LIN {X -0.331,Y -633.573,Z 342.601,A 0.000,B 0.000,C 90.000,E1 324.276} C_DIS
LIN {X 0.162,Y -638.117,Z 342.593,A 0.000,B 0.000,C 90.000,E1 322.718} C_DIS
LIN {X 0.137,Y -643.220,Z 342.583,A 0.000,B 0.000,C 90.000,E1 320.964} C_DIS
LIN {X 0.220,Y -647.759,Z 342.575,A 0.000,B 0.000,C 90.000,E1 319.461} C_DIS
LIN {X -0.093,Y -652.321,Z 342.567,A 0.000,B 0.000,C 90.000,E1 318.000} C_DIS
LIN {X 0.029,Y -660.222,Z 342.553,A 0.000,B 0.000,C 90.000,E1 315.526} C_DIS
LIN {X 0.410,Y -664.075,Z 342.546,A 0.000,B 0.000,C 90.000,E1 314.271} C_DIS
LIN {X -0.075,Y -667.878,Z 342.539,A 0.000,B 0.000,C 90.000,E1 313.095} C_DIS
LIN {X 0.010,Y -672.343,Z 342.531,A 0.000,B 0.000,C 90.000,E1 311.634} C_DIS
LIN {X 0.178,Y -676.385,Z 342.523,A 0.000,B 0.000,C 90.000,E1 310.172} C_DIS
LIN {X -0.049,Y -679.539,Z 342.517,A 0.000,B 0.000,C 90.000,E1 308.991} C_DIS
LIN {X 0.163,Y -681.944,Z 342.511,A 0.000,B 0.000,C 90.000,E1 308.016} C_DIS
LIN {X -0.404,Y -684.576,Z 342.505,A 0.000,B 0.000,C 90.000,E1 306.870} C_DIS
LIN {X -0.003,Y -686.307,Z 342.499,A 0.000,B 0.000,C 90.000,E1 305.884} C_DIS
LIN {X -0.162,Y -687.495,Z 342.495,A 0.000,B 0.000,C 90.000,E1 305.185} C_DIS
LIN {X 0.079,Y -688.424,Z 342.491,A 0.000,B 0.000,C 90.000,E1 304.452} C_DIS
LIN {X -0.452,Y -689.214,Z 342.488,A 0.000,B 0.000,C 90.000,E1 303.785} C_DIS
LIN {X -0.225,Y -689.609,Z 342.485,A 0.000,B 0.000,C 90.000,E1 303.293} C_DIS
LIN {X 0.216,Y -689.941,Z 342.481,A 0.000,B 0.000,C 90.000,E1 302.546} C_DIS
LIN {X -0.289,Y -689.979,Z 342.477,A 0.000,B 0.000,C 90.000,E1 301.878} C_DIS
LIN {X -0.067,Y -689.884,Z 342.474,A 0.000,B 0.000,C 90.000,E1 301.386} C_DIS
LIN {X -0.349,Y -689.175,Z 342.469,A 0.000,B 0.000,C 90.000,E1 300.463} C_DIS
LIN {X 0.107,Y -688.694,Z 342.466,A 0.000,B 0.000,C 90.000,E1 299.951} C_DIS
LIN {X -0.069,Y -687.718,Z 342.463,A 0.000,B 0.000,C 90.000,E1 299.255} C_DIS
LIN {X 0.000,Y -686.587,Z 342.459,A 0.000,B 0.000,C 90.000,E1 298.537} C_DIS
LIN {X 0.177,Y -684.270,Z 342.452,A 0.000,B 0.000,C 90.000,E1 297.334} C_DIS
LIN {X -0.067,Y -681.100,Z 342.444,A 0.000,B 0.000,C 90.000,E1 295.924} C_DIS
LIN {X 0.042,Y -678.136,Z 342.437,A 0.000,B 0.000,C 90.000,E1 294.719} C_DIS
LIN {X 0.274,Y -674.479,Z 342.429,A 0.000,B 0.000,C 90.000,E1 293.259} C_DIS
LIN {X -0.100,Y -670.508,Z 342.421,A 0.000,B 0.000,C 90.000,E1 291.844} C_DIS
LIN {X 0.164,Y -664.072,Z 342.408,A 0.000,B 0.000,C 90.000,E1 289.396} C_DIS
LIN {X -0.126,Y -657.475,Z 342.393,A 0.000,B 0.000,C 90.000,E1 286.732} C_DIS
LIN {X -0.104,Y -653.677,Z 342.383,A 0.000,B 0.000,C 90.000,E1 285.009} C_DIS
LIN {X -0.081,Y -648.752,Z 342.370,A 0.000,B 0.000,C 90.000,E1 282.535} C_DIS
LIN {X 0.182,Y -643.588,Z 342.350,A 0.000,B 0.000,C 90.000,E1 279.029} C_DIS
LIN {X 0.176,Y -640.607,Z 342.334,A 0.000,B 0.000,C 90.000,E1 276.030} C_DIS
LIN {X -0.117,Y -639.523,Z 342.324,A 0.000,B 0.000,C 90.000,E1 274.302} C_DIS
LIN {X -0.028,Y -638.474,Z 342.306,A 0.000,B 0.000,C 90.000,E1 271.031} C_DIS
LIN {X -0.005,Y -638.759,Z 342.288,A 0.000,B 0.000,C 90.000,E1 267.764} C_DIS
LIN {X -0.239,Y -639.730,Z 342.275,A 0.000,B 0.000,C 90.000,E1 265.527} C_DIS
LIN {X -0.105,Y -640.384,Z 342.268,A 0.000,B 0.000,C 90.000,E1 264.261} C_DIS
LIN {X 0.036,Y -641.104,Z 342.261,A 0.000,B 0.000,C 90.000,E1 262.996} C_DIS
LIN {X -0.074,Y -642.387,Z 342.251,A 0.000,B 0.000,C 90.000,E1 261.254} C_DIS
LIN {X -0.140,Y -643.675,Z 342.242,A 0.000,B 0.000,C 90.000,E1 259.511} C_DIS
LIN {X 0.137,Y -646.194,Z 342.228,A 0.000,B 0.000,C 90.000,E1 256.992} C_DIS
LIN {X 0.201,Y -647.266,Z 342.222,A 0.000,B 0.000,C 90.000,E1 255.992} C_DIS
LIN {X -0.214,Y -647.912,Z 342.218,A 0.000,B 0.000,C 90.000,E1 255.283} C_DIS
LIN {X -0.001,Y -648.296,Z 342.214,A 0.000,B 0.000,C 90.000,E1 254.519} C_DIS
LIN {X -0.100,Y -648.426,Z 342.211,A 0.000,B 0.000,C 90.000,E1 254.031} C_DIS
LIN {X -0.235,Y -648.404,Z 342.210,A 0.000,B 0.000,C 90.000,E1 253.795} C_DIS
LIN {X 0.249,Y -648.544,Z 342.209,A 0.000,B 0.000,C 90.000,E1 253.504} C_DIS
LIN {X 0.022,Y -648.427,Z 342.204,A 0.000,B 0.000,C 90.000,E1 252.779} C_DIS
LIN {X -0.259,Y -648.310,Z 342.202,A 0.000,B 0.000,C 90.000,E1 252.308} C_DIS
LIN {X 0.189,Y -647.802,Z 342.196,A 0.000,B 0.000,C 90.000,E1 251.275} C_DIS
LIN {X -0.043,Y -647.063,Z 342.192,A 0.000,B 0.000,C 90.000,E1 250.550} C_DIS
LIN {X -0.062,Y -645.989,Z 342.188,A 0.000,B 0.000,C 90.000,E1 249.806} C_DIS
LIN {X -0.312,Y -644.582,Z 342.184,A 0.000,B 0.000,C 90.000,E1 249.082} C_DIS
LIN {X 0.187,Y -643.530,Z 342.181,A 0.000,B 0.000,C 90.000,E1 248.539} C_DIS
LIN {X 0.137,Y -641.618,Z 342.177,A 0.000,B 0.000,C 90.000,E1 247.794} C_DIS
LIN {X 0.129,Y -638.725,Z 342.171,A 0.000,B 0.000,C 90.000,E1 246.794} C_DIS
LIN {X 0.132,Y -634.840,Z 342.164,A 0.000,B 0.000,C 90.000,E1 245.537} C_DIS
LIN {X 0.032,Y -631.434,Z 342.159,A 0.000,B 0.000,C 90.000,E1 244.537} C_DIS
LIN {X 0.178,Y -626.813,Z 342.152,A 0.000,B 0.000,C 90.000,E1 243.256} C_DIS
LIN {X -0.301,Y -620.193,Z 342.142,A 0.000,B 0.000,C 90.000,E1 241.513} C_DIS
LIN {X -0.080,Y -614.551,Z 342.133,A 0.000,B 0.000,C 90.000,E1 239.950} C_DIS
LIN {X -0.201,Y -608.779,Z 342.124,A 0.000,B 0.000,C 90.000,E1 238.408} C_DIS
LIN {X -0.038,Y -603.976,Z 342.117,A 0.000,B 0.000,C 90.000,E1 237.089} C_DIS
LIN {X 0.308,Y -600.039,Z 342.111,A 0.000,B 0.000,C 90.000,E1 236.008} C_DIS
LIN {X 0.039,Y -591.736,Z 342.098,A 0.000,B 0.000,C 90.000,E1 233.657} C_DIS
LIN {X 0.199,Y -588.943,Z 342.094,A 0.000,B 0.000,C 90.000,E1 232.844} C_DIS
LIN {X -0.190,Y -581.991,Z 342.083,A 0.000,B 0.000,C 90.000,E1 231.009} C_DIS
LIN {X 0.014,Y -572.772,Z 342.068,A 0.000,B 0.000,C 90.000,E1 228.286} C_DIS
LIN {X -0.123,Y -567.372,Z 342.059,A 0.000,B 0.000,C 90.000,E1 226.662} C_DIS
LIN {X 0.008,Y -561.901,Z 342.050,A 0.000,B 0.000,C 90.000,E1 225.000} C_DIS
LIN {X -0.045,Y -557.398,Z 342.042,A 0.000,B 0.000,C 90.000,E1 223.623} C_DIS
LIN {X 0.274,Y -552.030,Z 342.033,A 0.000,B 0.000,C 90.000,E1 221.919} C_DIS
LIN {X 0.115,Y -546.659,Z 342.024,A 0.000,B 0.000,C 90.000,E1 220.253} C_DIS
LIN {X -0.137,Y -540.630,Z 342.013,A 0.000,B 0.000,C 90.000,E1 218.302} C_DIS
LIN {X -0.034,Y -532.260,Z 341.997,A 0.000,B 0.000,C 90.000,E1 215.438} C_DIS
LIN {X -0.018,Y -526.719,Z 341.986,A 0.000,B 0.000,C 90.000,E1 213.420} C_DIS
LIN {X 0.007,Y -521.692,Z 341.974,A 0.000,B 0.000,C 90.000,E1 211.386} C_DIS
LIN {X 0.047,Y -518.302,Z 341.966,A 0.000,B 0.000,C 90.000,E1 209.922} C_DIS
LIN {X 0.126,Y -514.337,Z 341.957,A 0.000,B 0.000,C 90.000,E1 208.153} C_DIS
LIN {X -0.123,Y -510.480,Z 341.947,A 0.000,B 0.000,C 90.000,E1 206.411} C_DIS
LIN {X -0.221,Y -506.643,Z 341.937,A 0.000,B 0.000,C 90.000,E1 204.643} C_DIS
LIN {X 0.056,Y -502.697,Z 341.927,A 0.000,B 0.000,C 90.000,E1 202.823} C_DIS
LIN {X -0.139,Y -498.642,Z 341.917,A 0.000,B 0.000,C 90.000,E1 201.046} C_DIS
LIN {X 0.098,Y -493.870,Z 341.905,A 0.000,B 0.000,C 90.000,E1 198.906} C_DIS
LIN {X -0.090,Y -488.651,Z 341.892,A 0.000,B 0.000,C 90.000,E1 196.496} C_DIS
LIN {X 0.026,Y -485.563,Z 341.883,A 0.000,B 0.000,C 90.000,E1 194.954} C_DIS
LIN {X -0.188,Y -481.511,Z 341.871,A 0.000,B 0.000,C 90.000,E1 192.827} C_DIS
LIN {X -0.152,Y -477.561,Z 341.859,A 0.000,B 0.000,C 90.000,E1 190.658} C_DIS
LIN {X 0.203,Y -472.673,Z 341.844,A 0.000,B 0.000,C 90.000,E1 187.814} C_DIS
LIN {X 0.174,Y -469.159,Z 341.831,A 0.000,B 0.000,C 90.000,E1 185.625} C_DIS
LIN {X 0.005,Y -464.480,Z 341.812,A 0.000,B 0.000,C 90.000,E1 182.178} C_DIS
LIN {X -0.202,Y -460.613,Z 341.791,A 0.000,B 0.000,C 90.000,E1 178.396} C_DIS
LIN {X 0.167,Y -458.206,Z 341.768,A 0.000,B 0.000,C 90.000,E1 174.204} C_DIS
LIN {X -0.219,Y -457.795,Z 341.748,A 0.000,B 0.000,C 90.000,E1 170.735} C_DIS
LIN {X 0.146,Y -458.483,Z 341.725,A 0.000,B 0.000,C 90.000,E1 166.533} C_DIS
LIN {X -0.018,Y -460.753,Z 341.704,A 0.000,B 0.000,C 90.000,E1 162.725} C_DIS
LIN {X 0.071,Y -464.544,Z 341.683,A 0.000,B 0.000,C 90.000,E1 158.901} C_DIS
LIN {X 0.193,Y -467.993,Z 341.669,A 0.000,B 0.000,C 90.000,E1 156.357} C_DIS
LIN {X 0.134,Y -475.816,Z 341.644,A 0.000,B 0.000,C 90.000,E1 151.975} C_DIS
LIN {X -0.254,Y -485.313,Z 341.622,A 0.000,B 0.000,C 90.000,E1 147.995} C_DIS
LIN {X 0.261,Y -493.216,Z 341.607,A 0.000,B 0.000,C 90.000,E1 145.182} C_DIS
LIN {X -0.193,Y -498.805,Z 341.597,A 0.000,B 0.000,C 90.000,E1 143.417} C_DIS
LIN {X -0.230,Y -504.475,Z 341.587,A 0.000,B 0.000,C 90.000,E1 141.618} C_DIS
LIN {X -0.022,Y -507.950,Z 341.580,A 0.000,B 0.000,C 90.000,E1 140.400} C_DIS
LIN {X -0.223,Y -509.634,Z 341.577,A 0.000,B 0.000,C 90.000,E1 139.828} C_DIS
LIN {X -0.019,Y -513.555,Z 341.569,A 0.000,B 0.000,C 90.000,E1 138.324} C_DIS
LIN {X -0.316,Y -515.644,Z 341.564,A 0.000,B 0.000,C 90.000,E1 137.472} C_DIS
LIN {X 0.137,Y -517.338,Z 341.559,A 0.000,B 0.000,C 90.000,E1 136.539} C_DIS
LIN {X 0.238,Y -518.689,Z 341.554,A 0.000,B 0.000,C 90.000,E1 135.648} C_DIS
LIN {X -0.013,Y -519.734,Z 341.549,A 0.000,B 0.000,C 90.000,E1 134.798} C_DIS
LIN {X -0.252,Y -520.479,Z 341.544,A 0.000,B 0.000,C 90.000,E1 133.947} C_DIS
LIN {X -0.119,Y -520.772,Z 341.539,A 0.000,B 0.000,C 90.000,E1 133.056} C_DIS
LIN {X 0.044,Y -520.897,Z 341.534,A 0.000,B 0.000,C 90.000,E1 132.162} C_DIS
LIN {X 0.112,Y -520.488,Z 341.528,A 0.000,B 0.000,C 90.000,E1 130.987} C_DIS
LIN {X 0.281,Y -519.807,Z 341.523,A 0.000,B 0.000,C 90.000,E1 130.092} C_DIS
LIN {X -0.287,Y -518.859,Z 341.518,A 0.000,B 0.000,C 90.000,E1 129.277} C_DIS
LIN {X -0.319,Y -516.516,Z 341.508,A 0.000,B 0.000,C 90.000,E1 127.523} C_DIS
LIN {X 0.141,Y -514.956,Z 341.502,A 0.000,B 0.000,C 90.000,E1 126.297} C_DIS
LIN {X -0.149,Y -513.122,Z 341.495,A 0.000,B 0.000,C 90.000,E1 125.152} C_DIS
LIN {X -0.337,Y -511.198,Z 341.489,A 0.000,B 0.000,C 90.000,E1 123.992} C_DIS
LIN {X 0.158,Y -508.967,Z 341.482,A 0.000,B 0.000,C 90.000,E1 122.752} C_DIS
LIN {X 0.233,Y -505.879,Z 341.474,A 0.000,B 0.000,C 90.000,E1 121.258} C_DIS
LIN {X -0.013,Y -502.675,Z 341.466,A 0.000,B 0.000,C 90.000,E1 119.795} C_DIS
LIN {X -0.177,Y -500.003,Z 341.459,A 0.000,B 0.000,C 90.000,E1 118.615} C_DIS
LIN {X -0.017,Y -495.022,Z 341.447,A 0.000,B 0.000,C 90.000,E1 116.488} C_DIS
LIN {X 0.170,Y -491.271,Z 341.439,A 0.000,B 0.000,C 90.000,E1 114.951} C_DIS
LIN {X -0.179,Y -488.967,Z 341.434,A 0.000,B 0.000,C 90.000,E1 114.079} C_DIS
LIN {X 0.127,Y -484.863,Z 341.425,A 0.000,B 0.000,C 90.000,E1 112.514} C_DIS
LIN {X 0.164,Y -480.627,Z 341.417,A 0.000,B 0.000,C 90.000,E1 110.972} C_DIS
LIN {X -0.012,Y -478.861,Z 341.413,A 0.000,B 0.000,C 90.000,E1 110.375} C_DIS
LIN {X -0.070,Y -474.964,Z 341.406,A 0.000,B 0.000,C 90.000,E1 109.141} C_DIS
LIN {X 0.097,Y -470.837,Z 341.399,A 0.000,B 0.000,C 90.000,E1 107.873} C_DIS
LIN {X 0.061,Y -466.513,Z 341.392,A 0.000,B 0.000,C 90.000,E1 106.622} C_DIS
LIN {X -0.056,Y -464.782,Z 341.390,A 0.000,B 0.000,C 90.000,E1 106.134} C_DIS
LIN {X -0.096,Y -464.792,Z 341.390,A 0.000,B 0.000,C 90.000,E1 106.134} C_DIS
LIN {X -0.112,Y -467.396,Z 341.384,A 0.000,B 0.000,C 90.000,E1 105.064} C_DIS
LIN {X 0.144,Y -468.032,Z 341.382,A 0.000,B 0.000,C 90.000,E1 104.717} C_DIS
LIN {X 0.121,Y -476.242,Z 341.356,A 0.000,B 0.000,C 90.000,E1 100.018} C_DIS
LIN {X -0.093,Y -482.135,Z 341.330,A 0.000,B 0.000,C 90.000,E1 95.391} C_DIS
LIN {X 0.142,Y -485.531,Z 341.304,A 0.000,B 0.000,C 90.000,E1 90.745} C_DIS
LIN {X 0.174,Y -486.379,Z 341.280,A 0.000,B 0.000,C 90.000,E1 86.445} C_DIS
LIN {X -0.002,Y -486.347,Z 341.279,A 0.000,B 0.000,C 90.000,E1 86.159} C_DIS
LIN {X 0.077,Y -484.661,Z 341.253,A 0.000,B 0.000,C 90.000,E1 81.546} C_DIS
LIN {X -0.033,Y -480.580,Z 341.227,A 0.000,B 0.000,C 90.000,E1 76.937} C_DIS
LIN {X 0.114,Y -479.153,Z 341.222,A 0.000,B 0.000,C 90.000,E1 75.992} C_DIS
LIN {X -0.153,Y -477.278,Z 341.215,A 0.000,B 0.000,C 90.000,E1 74.755} C_DIS
LIN {X -0.193,Y -477.290,Z 341.215,A 0.000,B 0.000,C 90.000,E1 74.755} C_DIS
LIN {X 0.146,Y -479.250,Z 341.213,A 0.000,B 0.000,C 90.000,E1 74.283} C_DIS
LIN {X 0.188,Y -482.615,Z 341.209,A 0.000,B 0.000,C 90.000,E1 73.504} C_DIS
LIN {X 0.035,Y -486.200,Z 341.203,A 0.000,B 0.000,C 90.000,E1 72.598} C_DIS
LIN {X -0.097,Y -488.431,Z 341.200,A 0.000,B 0.000,C 90.000,E1 72.000} C_DIS
LIN {X -0.160,Y -492.635,Z 341.193,A 0.000,B 0.000,C 90.000,E1 70.786} C_DIS
LIN {X -0.161,Y -496.592,Z 341.186,A 0.000,B 0.000,C 90.000,E1 69.571} C_DIS
LIN {X 0.008,Y -499.421,Z 341.181,A 0.000,B 0.000,C 90.000,E1 68.646} C_DIS
LIN {X 0.097,Y -503.009,Z 341.175,A 0.000,B 0.000,C 90.000,E1 67.433} C_DIS
LIN {X 0.159,Y -506.550,Z 341.168,A 0.000,B 0.000,C 90.000,E1 66.230} C_DIS
LIN {X -0.290,Y -510.836,Z 341.160,A 0.000,B 0.000,C 90.000,E1 64.793} C_DIS
LIN {X -0.109,Y -515.891,Z 341.150,A 0.000,B 0.000,C 90.000,E1 62.999} C_DIS
LIN {X -0.275,Y -520.923,Z 341.140,A 0.000,B 0.000,C 90.000,E1 61.257} C_DIS
LIN {X 0.178,Y -525.883,Z 341.130,A 0.000,B 0.000,C 90.000,E1 59.459} C_DIS
LIN {X -0.119,Y -529.994,Z 341.122,A 0.000,B 0.000,C 90.000,E1 58.043} C_DIS
LIN {X 0.097,Y -533.975,Z 341.114,A 0.000,B 0.000,C 90.000,E1 56.580} C_DIS
LIN {X 0.079,Y -536.345,Z 341.110,A 0.000,B 0.000,C 90.000,E1 55.722} C_DIS
LIN {X 0.251,Y -540.067,Z 341.102,A 0.000,B 0.000,C 90.000,E1 54.276} C_DIS
LIN {X 0.335,Y -542.844,Z 341.095,A 0.000,B 0.000,C 90.000,E1 53.130} C_DIS
LIN {X 0.030,Y -545.366,Z 341.089,A 0.000,B 0.000,C 90.000,E1 52.029} C_DIS
LIN {X 0.148,Y -547.153,Z 341.084,A 0.000,B 0.000,C 90.000,E1 51.170} C_DIS
LIN {X -0.101,Y -549.343,Z 341.078,A 0.000,B 0.000,C 90.000,E1 50.070} C_DIS
LIN {X -0.018,Y -550.749,Z 341.073,A 0.000,B 0.000,C 90.000,E1 49.218} C_DIS
LIN {X -0.279,Y -551.972,Z 341.069,A 0.000,B 0.000,C 90.000,E1 48.405} C_DIS
LIN {X 0.192,Y -552.775,Z 341.066,A 0.000,B 0.000,C 90.000,E1 47.796} C_DIS
LIN {X -0.039,Y -553.939,Z 341.059,A 0.000,B 0.000,C 90.000,E1 46.701} C_DIS
LIN {X -0.306,Y -554.575,Z 341.055,A 0.000,B 0.000,C 90.000,E1 45.891} C_DIS
LIN {X -0.216,Y -554.911,Z 341.052,A 0.000,B 0.000,C 90.000,E1 45.324} C_DIS
LIN {X -0.029,Y -555.097,Z 341.046,A 0.000,B 0.000,C 90.000,E1 44.190} C_DIS
LIN {X 0.153,Y -554.835,Z 341.039,A 0.000,B 0.000,C 90.000,E1 43.056} C_DIS
LIN {X -0.055,Y -554.245,Z 341.033,A 0.000,B 0.000,C 90.000,E1 41.962} C_DIS
LIN {X 0.143,Y -553.352,Z 341.027,A 0.000,B 0.000,C 90.000,E1 40.825} C_DIS
LIN {X 0.034,Y -551.881,Z 341.019,A 0.000,B 0.000,C 90.000,E1 39.439} C_DIS
LIN {X 0.194,Y -550.558,Z 341.013,A 0.000,B 0.000,C 90.000,E1 38.302} C_DIS
LIN {X -0.138,Y -547.744,Z 341.000,A 0.000,B 0.000,C 90.000,E1 36.091} C_DIS
LIN {X -0.183,Y -545.658,Z 340.991,A 0.000,B 0.000,C 90.000,E1 34.405} C_DIS
LIN {X -0.071,Y -543.005,Z 340.979,A 0.000,B 0.000,C 90.000,E1 32.133} C_DIS
LIN {X 0.116,Y -540.842,Z 340.967,A 0.000,B 0.000,C 90.000,E1 30.129} C_DIS
LIN {X -0.012,Y -539.161,Z 340.958,A 0.000,B 0.000,C 90.000,E1 28.437} C_DIS
LIN {X -0.173,Y -537.406,Z 340.949,A 0.000,B 0.000,C 90.000,E1 26.744} C_DIS
LIN {X -0.210,Y -535.241,Z 340.936,A 0.000,B 0.000,C 90.000,E1 24.463} C_DIS
LIN {X 0.049,Y -533.722,Z 340.926,A 0.000,B 0.000,C 90.000,E1 22.717} C_DIS
LIN {X 0.267,Y -532.445,Z 340.917,A 0.000,B 0.000,C 90.000,E1 20.972} C_DIS
LIN {X 0.258,Y -531.235,Z 340.906,A 0.000,B 0.000,C 90.000,E1 18.960} C_DIS
LIN {X 0.092,Y -530.016,Z 340.891,A 0.000,B 0.000,C 90.000,E1 16.386} C_DIS
LIN {X -0.252,Y -529.180,Z 340.877,A 0.000,B 0.000,C 90.000,E1 13.828} C_DIS
LIN {X 0.119,Y -528.971,Z 340.864,A 0.000,B 0.000,C 90.000,E1 11.478} C_DIS
LIN {X -0.240,Y -529.318,Z 340.851,A 0.000,B 0.000,C 90.000,E1 9.208} C_DIS
LIN {X -0.186,Y -530.214,Z 340.837,A 0.000,B 0.000,C 90.000,E1 6.606} C_DIS
LIN {X -0.167,Y -530.972,Z 340.829,A 0.000,B 0.000,C 90.000,E1 5.163} C_DIS
LIN {X -0.222,Y -533.580,Z 340.809,A 0.000,B 0.000,C 90.000,E1 1.718} C_DIS
LIN {X 0.216,Y -536.762,Z 340.793,A 0.000,B 0.000,C 90.000,E1 358.625} C_DIS
LIN {X 0.261,Y -538.239,Z 340.786,A 0.000,B 0.000,C 90.000,E1 357.478} C_DIS
LIN {X -0.147,Y -540.742,Z 340.777,A 0.000,B 0.000,C 90.000,E1 355.812} C_DIS
LIN {X 0.018,Y -542.712,Z 340.769,A 0.000,B 0.000,C 90.000,E1 354.375} C_DIS
LIN {X 0.274,Y -544.976,Z 340.761,A 0.000,B 0.000,C 90.000,E1 352.932} C_DIS
LIN {X 0.248,Y -549.580,Z 340.748,A 0.000,B 0.000,C 90.000,E1 350.679} C_DIS
LIN {X 0.100,Y -555.281,Z 340.734,A 0.000,B 0.000,C 90.000,E1 348.173} C_DIS
LIN {X 0.234,Y -561.591,Z 340.722,A 0.000,B 0.000,C 90.000,E1 345.936} C_DIS
LIN {X 0.095,Y -569.770,Z 340.707,A 0.000,B 0.000,C 90.000,E1 343.196} C_DIS
LIN {X 0.216,Y -574.145,Z 340.699,A 0.000,B 0.000,C 90.000,E1 341.819} C_DIS
LIN {X 0.235,Y -579.315,Z 340.690,A 0.000,B 0.000,C 90.000,E1 340.188} C_DIS
LIN {X 0.153,Y -583.628,Z 340.683,A 0.000,B 0.000,C 90.000,E1 338.847} C_DIS
LIN {X 0.235,Y -588.795,Z 340.674,A 0.000,B 0.000,C 90.000,E1 337.230} C_DIS
LIN {X -0.010,Y -593.190,Z 340.666,A 0.000,B 0.000,C 90.000,E1 335.921} C_DIS
LIN {X -0.098,Y -599.562,Z 340.656,A 0.000,B 0.000,C 90.000,E1 334.076} C_DIS
LIN {X 0.025,Y -605.068,Z 340.647,A 0.000,B 0.000,C 90.000,E1 332.487} C_DIS
LIN {X -0.002,Y -610.599,Z 340.639,A 0.000,B 0.000,C 90.000,E1 330.923} C_DIS
LIN {X -0.169,Y -617.246,Z 340.628,A 0.000,B 0.000,C 90.000,E1 329.125} C_DIS
LIN {X 0.371,Y -621.878,Z 340.621,A 0.000,B 0.000,C 90.000,E1 327.788} C_DIS
LIN {X -0.062,Y -626.310,Z 340.614,A 0.000,B 0.000,C 90.000,E1 326.548} C_DIS
LIN {X -0.253,Y -628.841,Z 340.610,A 0.000,B 0.000,C 90.000,E1 325.801} C_DIS
LIN {X -0.217,Y -633.664,Z 340.601,A 0.000,B 0.000,C 90.000,E1 324.276} C_DIS
LIN {X -0.229,Y -638.199,Z 340.593,A 0.000,B 0.000,C 90.000,E1 322.763} C_DIS
LIN {X -0.244,Y -643.292,Z 340.583,A 0.000,B 0.000,C 90.000,E1 321.009} C_DIS
LIN {X 0.342,Y -647.820,Z 340.575,A 0.000,B 0.000,C 90.000,E1 319.461} C_DIS
LIN {X -0.019,Y -653.071,Z 340.565,A 0.000,B 0.000,C 90.000,E1 317.757} C_DIS
LIN {X -0.316,Y -660.190,Z 340.553,A 0.000,B 0.000,C 90.000,E1 315.567} C_DIS
LIN {X -0.403,Y -664.044,Z 340.546,A 0.000,B 0.000,C 90.000,E1 314.352} C_DIS
LIN {X 0.051,Y -667.807,Z 340.539,A 0.000,B 0.000,C 90.000,E1 313.095} C_DIS
LIN {X -0.367,Y -672.208,Z 340.531,A 0.000,B 0.000,C 90.000,E1 311.676} C_DIS
LIN {X 0.301,Y -676.198,Z 340.523,A 0.000,B 0.000,C 90.000,E1 310.172} C_DIS
LIN {X 0.071,Y -679.245,Z 340.517,A 0.000,B 0.000,C 90.000,E1 308.991} C_DIS
LIN {X 0.254,Y -681.060,Z 340.513,A 0.000,B 0.000,C 90.000,E1 308.257} C_DIS
LIN {X -0.293,Y -684.167,Z 340.505,A 0.000,B 0.000,C 90.000,E1 306.870} C_DIS
LIN {X 0.128,Y -686.232,Z 340.498,A 0.000,B 0.000,C 90.000,E1 305.644} C_DIS
LIN {X -0.061,Y -686.985,Z 340.495,A 0.000,B 0.000,C 90.000,E1 305.185} C_DIS
LIN {X -0.213,Y -687.857,Z 340.492,A 0.000,B 0.000,C 90.000,E1 304.485} C_DIS
LIN {X -0.360,Y -688.586,Z 340.488,A 0.000,B 0.000,C 90.000,E1 303.785} C_DIS
LIN {X -0.137,Y -688.969,Z 340.485,A 0.000,B 0.000,C 90.000,E1 303.293} C_DIS
LIN {X 0.297,Y -689.226,Z 340.481,A 0.000,B 0.000,C 90.000,E1 302.546} C_DIS
LIN {X -0.214,Y -689.196,Z 340.477,A 0.000,B 0.000,C 90.000,E1 301.878} C_DIS
LIN {X 0.002,Y -689.063,Z 340.474,A 0.000,B 0.000,C 90.000,E1 301.386} C_DIS
LIN {X 0.080,Y -688.534,Z 340.470,A 0.000,B 0.000,C 90.000,E1 300.669} C_DIS
LIN {X 0.161,Y -687.814,Z 340.467,A 0.000,B 0.000,C 90.000,E1 299.951} C_DIS
LIN {X -0.360,Y -686.820,Z 340.463,A 0.000,B 0.000,C 90.000,E1 299.283} C_DIS
LIN {X -0.291,Y -685.647,Z 340.459,A 0.000,B 0.000,C 90.000,E1 298.565} C_DIS
LIN {X 0.198,Y -683.267,Z 340.452,A 0.000,B 0.000,C 90.000,E1 297.334} C_DIS
LIN {X 0.029,Y -680.586,Z 340.445,A 0.000,B 0.000,C 90.000,E1 296.155} C_DIS
LIN {X -0.077,Y -678.288,Z 340.440,A 0.000,B 0.000,C 90.000,E1 295.207} C_DIS
LIN {X -0.118,Y -674.603,Z 340.432,A 0.000,B 0.000,C 90.000,E1 293.770} C_DIS
LIN {X 0.149,Y -672.697,Z 340.428,A 0.000,B 0.000,C 90.000,E1 293.025} C_DIS
LIN {X -0.002,Y -668.678,Z 340.420,A 0.000,B 0.000,C 90.000,E1 291.589} C_DIS
LIN {X 0.071,Y -662.878,Z 340.408,A 0.000,B 0.000,C 90.000,E1 289.396} C_DIS
LIN {X -0.232,Y -657.422,Z 340.396,A 0.000,B 0.000,C 90.000,E1 287.221} C_DIS
LIN {X -0.145,Y -653.011,Z 340.385,A 0.000,B 0.000,C 90.000,E1 285.245} C_DIS
LIN {X -0.280,Y -647.584,Z 340.370,A 0.000,B 0.000,C 90.000,E1 282.535} C_DIS
LIN {X 0.094,Y -642.728,Z 340.352,A 0.000,B 0.000,C 90.000,E1 279.265} C_DIS
LIN {X -0.121,Y -639.457,Z 340.333,A 0.000,B 0.000,C 90.000,E1 276.030} C_DIS
LIN {X 0.198,Y -638.381,Z 340.324,A 0.000,B 0.000,C 90.000,E1 274.245} C_DIS
LIN {X 0.240,Y -637.343,Z 340.306,A 0.000,B 0.000,C 90.000,E1 270.974} C_DIS
LIN {X 0.213,Y -637.644,Z 340.287,A 0.000,B 0.000,C 90.000,E1 267.707} C_DIS
LIN {X -0.054,Y -638.621,Z 340.275,A 0.000,B 0.000,C 90.000,E1 265.469} C_DIS
LIN {X 0.061,Y -639.278,Z 340.268,A 0.000,B 0.000,C 90.000,E1 264.204} C_DIS
LIN {X -0.194,Y -639.914,Z 340.262,A 0.000,B 0.000,C 90.000,E1 263.223} C_DIS
LIN {X 0.046,Y -641.363,Z 340.251,A 0.000,B 0.000,C 90.000,E1 261.197} C_DIS
LIN {X 0.114,Y -642.542,Z 340.243,A 0.000,B 0.000,C 90.000,E1 259.690} C_DIS
LIN {X 0.196,Y -645.387,Z 340.228,A 0.000,B 0.000,C 90.000,E1 256.937} C_DIS
LIN {X 0.246,Y -646.485,Z 340.222,A 0.000,B 0.000,C 90.000,E1 255.936} C_DIS
LIN {X -0.178,Y -647.247,Z 340.218,A 0.000,B 0.000,C 90.000,E1 255.227} C_DIS
LIN {X 0.166,Y -647.567,Z 340.215,A 0.000,B 0.000,C 90.000,E1 254.700} C_DIS
LIN {X -0.357,Y -648.061,Z 340.208,A 0.000,B 0.000,C 90.000,E1 253.504} C_DIS
LIN {X 0.030,Y -648.088,Z 340.204,A 0.000,B 0.000,C 90.000,E1 252.725} C_DIS
LIN {X -0.342,Y -647.947,Z 340.199,A 0.000,B 0.000,C 90.000,E1 251.764} C_DIS
LIN {X 0.250,Y -647.464,Z 340.194,A 0.000,B 0.000,C 90.000,E1 250.967} C_DIS
LIN {X -0.049,Y -647.000,Z 340.192,A 0.000,B 0.000,C 90.000,E1 250.496} C_DIS
LIN {X -0.071,Y -645.909,Z 340.188,A 0.000,B 0.000,C 90.000,E1 249.752} C_DIS
LIN {X -0.325,Y -644.594,Z 340.183,A 0.000,B 0.000,C 90.000,E1 249.028} C_DIS
LIN {X 0.299,Y -642.408,Z 340.178,A 0.000,B 0.000,C 90.000,E1 247.975} C_DIS
LIN {X 0.242,Y -640.412,Z 340.174,A 0.000,B 0.000,C 90.000,E1 247.230} C_DIS
LIN {X 0.108,Y -639.072,Z 340.171,A 0.000,B 0.000,C 90.000,E1 246.741} C_DIS
LIN {X 0.112,Y -635.371,Z 340.164,A 0.000,B 0.000,C 90.000,E1 245.485} C_DIS
LIN {X 0.287,Y -632.038,Z 340.158,A 0.000,B 0.000,C 90.000,E1 244.460} C_DIS
LIN {X 0.141,Y -628.439,Z 340.153,A 0.000,B 0.000,C 90.000,E1 243.461} C_DIS
LIN {X -0.352,Y -625.674,Z 340.148,A 0.000,B 0.000,C 90.000,E1 242.743} C_DIS
LIN {X -0.015,Y -619.156,Z 340.139,A 0.000,B 0.000,C 90.000,E1 240.923} C_DIS
LIN {X 0.233,Y -615.503,Z 340.133,A 0.000,B 0.000,C 90.000,E1 239.871} C_DIS
LIN {X 0.134,Y -609.825,Z 340.124,A 0.000,B 0.000,C 90.000,E1 238.329} C_DIS
LIN {X -0.012,Y -605.061,Z 340.117,A 0.000,B 0.000,C 90.000,E1 237.041} C_DIS
LIN {X -0.407,Y -602.162,Z 340.113,A 0.000,B 0.000,C 90.000,E1 236.294} C_DIS
LIN {X -0.033,Y -592.817,Z 340.098,A 0.000,B 0.000,C 90.000,E1 233.623} C_DIS
LIN {X -0.211,Y -589.997,Z 340.094,A 0.000,B 0.000,C 90.000,E1 232.844} C_DIS
LIN {X -0.116,Y -583.100,Z 340.083,A 0.000,B 0.000,C 90.000,E1 230.964} C_DIS
LIN {X -0.035,Y -574.757,Z 340.070,A 0.000,B 0.000,C 90.000,E1 228.528} C_DIS
LIN {X 0.166,Y -570.277,Z 340.062,A 0.000,B 0.000,C 90.000,E1 227.148} C_DIS
LIN {X 0.174,Y -566.651,Z 340.056,A 0.000,B 0.000,C 90.000,E1 226.053} C_DIS
LIN {X -0.118,Y -561.213,Z 340.047,A 0.000,B 0.000,C 90.000,E1 224.433} C_DIS
LIN {X -0.119,Y -555.783,Z 340.038,A 0.000,B 0.000,C 90.000,E1 222.771} C_DIS
LIN {X 0.112,Y -551.307,Z 340.030,A 0.000,B 0.000,C 90.000,E1 221.353} C_DIS
LIN {X -0.032,Y -545.133,Z 340.019,A 0.000,B 0.000,C 90.000,E1 219.402} C_DIS
LIN {X 0.136,Y -540.846,Z 340.011,A 0.000,B 0.000,C 90.000,E1 217.971} C_DIS
LIN {X -0.172,Y -533.358,Z 339.997,A 0.000,B 0.000,C 90.000,E1 215.438} C_DIS
LIN {X -0.066,Y -525.632,Z 339.981,A 0.000,B 0.000,C 90.000,E1 212.546} C_DIS
LIN {X 0.054,Y -520.062,Z 339.968,A 0.000,B 0.000,C 90.000,E1 210.207} C_DIS
LIN {X 0.090,Y -515.411,Z 339.957,A 0.000,B 0.000,C 90.000,E1 208.153} C_DIS
LIN {X -0.018,Y -512.195,Z 339.948,A 0.000,B 0.000,C 90.000,E1 206.693} C_DIS
LIN {X -0.211,Y -507.715,Z 339.937,A 0.000,B 0.000,C 90.000,E1 204.643} C_DIS
LIN {X 0.091,Y -503.755,Z 339.927,A 0.000,B 0.000,C 90.000,E1 202.823} C_DIS
LIN {X -0.156,Y -500.414,Z 339.919,A 0.000,B 0.000,C 90.000,E1 201.354} C_DIS
LIN {X 0.184,Y -496.984,Z 339.910,A 0.000,B 0.000,C 90.000,E1 199.812} C_DIS
LIN {X 0.121,Y -493.646,Z 339.902,A 0.000,B 0.000,C 90.000,E1 198.308} C_DIS
LIN {X 0.028,Y -489.774,Z 339.892,A 0.000,B 0.000,C 90.000,E1 196.496} C_DIS
LIN {X -0.183,Y -487.346,Z 339.885,A 0.000,B 0.000,C 90.000,E1 195.300} C_DIS
LIN {X -0.020,Y -482.665,Z 339.871,A 0.000,B 0.000,C 90.000,E1 192.827} C_DIS
LIN {X 0.047,Y -478.750,Z 339.859,A 0.000,B 0.000,C 90.000,E1 190.658} C_DIS
LIN {X -0.169,Y -474.868,Z 339.847,A 0.000,B 0.000,C 90.000,E1 188.511} C_DIS
LIN {X -0.137,Y -472.343,Z 339.839,A 0.000,B 0.000,C 90.000,E1 186.947} C_DIS
LIN {X -0.179,Y -468.092,Z 339.823,A 0.000,B 0.000,C 90.000,E1 184.131} C_DIS
LIN {X 0.080,Y -465.307,Z 339.811,A 0.000,B 0.000,C 90.000,E1 181.892} C_DIS
LIN {X 0.165,Y -461.833,Z 339.791,A 0.000,B 0.000,C 90.000,E1 178.396} C_DIS
LIN {X 0.094,Y -459.211,Z 339.765,A 0.000,B 0.000,C 90.000,E1 173.628} C_DIS
LIN {X -0.197,Y -458.964,Z 339.749,A 0.000,B 0.000,C 90.000,E1 170.792} C_DIS
LIN {X -0.213,Y -459.596,Z 339.726,A 0.000,B 0.000,C 90.000,E1 166.645} C_DIS
LIN {X -0.095,Y -462.009,Z 339.703,A 0.000,B 0.000,C 90.000,E1 162.489} C_DIS
LIN {X 0.105,Y -465.470,Z 339.683,A 0.000,B 0.000,C 90.000,E1 158.975} C_DIS
LIN {X -0.238,Y -469.343,Z 339.668,A 0.000,B 0.000,C 90.000,E1 156.177} C_DIS
LIN {X -0.019,Y -477.234,Z 339.643,A 0.000,B 0.000,C 90.000,E1 151.769} C_DIS
LIN {X 0.080,Y -486.801,Z 339.621,A 0.000,B 0.000,C 90.000,E1 147.740} C_DIS
LIN {X 0.233,Y -494.691,Z 339.606,A 0.000,B 0.000,C 90.000,E1 144.975} C_DIS
LIN {X -0.190,Y -500.189,Z 339.596,A 0.000,B 0.000,C 90.000,E1 143.210} C_DIS
LIN {X -0.088,Y -504.817,Z 339.587,A 0.000,B 0.000,C 90.000,E1 141.698} C_DIS
LIN {X 0.023,Y -509.062,Z 339.579,A 0.000,B 0.000,C 90.000,E1 140.194} C_DIS
LIN {X -0.026,Y -512.139,Z 339.572,A 0.000,B 0.000,C 90.000,E1 139.013} C_DIS
LIN {X 0.043,Y -514.354,Z 339.567,A 0.000,B 0.000,C 90.000,E1 138.119} C_DIS
LIN {X 0.101,Y -516.219,Z 339.563,A 0.000,B 0.000,C 90.000,E1 137.229} C_DIS
LIN {X -0.087,Y -517.293,Z 339.559,A 0.000,B 0.000,C 90.000,E1 136.662} C_DIS
LIN {X 0.027,Y -518.564,Z 339.554,A 0.000,B 0.000,C 90.000,E1 135.769} C_DIS
LIN {X -0.230,Y -519.563,Z 339.549,A 0.000,B 0.000,C 90.000,E1 134.919} C_DIS
LIN {X -0.103,Y -520.287,Z 339.545,A 0.000,B 0.000,C 90.000,E1 134.028} C_DIS
LIN {X -0.038,Y -520.598,Z 339.538,A 0.000,B 0.000,C 90.000,E1 132.852} C_DIS
LIN {X -0.258,Y -520.624,Z 339.533,A 0.000,B 0.000,C 90.000,E1 132.000} C_DIS
LIN {X 0.255,Y -520.170,Z 339.528,A 0.000,B 0.000,C 90.000,E1 131.067} C_DIS
LIN {X -0.035,Y -519.066,Z 339.522,A 0.000,B 0.000,C 90.000,E1 129.930} C_DIS
LIN {X 0.117,Y -518.019,Z 339.517,A 0.000,B 0.000,C 90.000,E1 129.036} C_DIS
LIN {X -0.192,Y -516.041,Z 339.509,A 0.000,B 0.000,C 90.000,E1 127.604} C_DIS
LIN {X 0.192,Y -514.021,Z 339.501,A 0.000,B 0.000,C 90.000,E1 126.091} C_DIS
LIN {X -0.110,Y -512.167,Z 339.494,A 0.000,B 0.000,C 90.000,E1 124.945} C_DIS
LIN {X 0.061,Y -510.724,Z 339.489,A 0.000,B 0.000,C 90.000,E1 124.040} C_DIS
LIN {X 0.168,Y -507.928,Z 339.481,A 0.000,B 0.000,C 90.000,E1 122.546} C_DIS
LIN {X -0.039,Y -504.824,Z 339.473,A 0.000,B 0.000,C 90.000,E1 121.082} C_DIS
LIN {X -0.047,Y -501.597,Z 339.464,A 0.000,B 0.000,C 90.000,E1 119.589} C_DIS
LIN {X 0.210,Y -498.952,Z 339.458,A 0.000,B 0.000,C 90.000,E1 118.359} C_DIS
LIN {X -0.102,Y -494.042,Z 339.446,A 0.000,B 0.000,C 90.000,E1 116.283} C_DIS
LIN {X -0.146,Y -490.375,Z 339.438,A 0.000,B 0.000,C 90.000,E1 114.771} C_DIS
LIN {X 0.144,Y -488.095,Z 339.432,A 0.000,B 0.000,C 90.000,E1 113.823} C_DIS
LIN {X -0.204,Y -484.093,Z 339.424,A 0.000,B 0.000,C 90.000,E1 112.333} C_DIS
LIN {X -0.175,Y -480.776,Z 339.417,A 0.000,B 0.000,C 90.000,E1 111.099} C_DIS
LIN {X -0.181,Y -479.111,Z 339.414,A 0.000,B 0.000,C 90.000,E1 110.482} C_DIS
LIN {X 0.028,Y -474.413,Z 339.405,A 0.000,B 0.000,C 90.000,E1 108.906} C_DIS
LIN {X 0.189,Y -470.422,Z 339.398,A 0.000,B 0.000,C 90.000,E1 107.638} C_DIS
LIN {X -0.104,Y -467.402,Z 339.393,A 0.000,B 0.000,C 90.000,E1 106.732} C_DIS
LIN {X -0.030,Y -465.041,Z 339.389,A 0.000,B 0.000,C 90.000,E1 106.024} C_DIS
LIN {X -0.070,Y -465.043,Z 339.389,A 0.000,B 0.000,C 90.000,E1 106.024} C_DIS
LIN {X -0.019,Y -467.904,Z 339.382,A 0.000,B 0.000,C 90.000,E1 104.828} C_DIS
LIN {X 0.009,Y -475.472,Z 339.358,A 0.000,B 0.000,C 90.000,E1 100.433} C_DIS
LIN {X -0.153,Y -476.118,Z 339.356,A 0.000,B 0.000,C 90.000,E1 100.141} C_DIS
LIN {X 0.130,Y -482.036,Z 339.330,A 0.000,B 0.000,C 90.000,E1 95.454} C_DIS
LIN {X -0.079,Y -485.470,Z 339.305,A 0.000,B 0.000,C 90.000,E1 90.859} C_DIS
LIN {X -0.149,Y -485.574,Z 339.295,A 0.000,B 0.000,C 90.000,E1 89.026} C_DIS
LIN {X -0.046,Y -486.385,Z 339.281,A 0.000,B 0.000,C 90.000,E1 86.560} C_DIS
LIN {X -0.221,Y -486.364,Z 339.279,A 0.000,B 0.000,C 90.000,E1 86.274} C_DIS
LIN {X -0.133,Y -484.690,Z 339.254,A 0.000,B 0.000,C 90.000,E1 81.659} C_DIS
LIN {X -0.118,Y -483.700,Z 339.249,A 0.000,B 0.000,C 90.000,E1 80.735} C_DIS
LIN {X 0.246,Y -480.628,Z 339.228,A 0.000,B 0.000,C 90.000,E1 76.992} C_DIS
LIN {X 0.103,Y -480.311,Z 339.226,A 0.000,B 0.000,C 90.000,E1 76.700} C_DIS
LIN {X -0.192,Y -477.347,Z 339.216,A 0.000,B 0.000,C 90.000,E1 74.810} C_DIS
LIN {X -0.233,Y -477.360,Z 339.216,A 0.000,B 0.000,C 90.000,E1 74.810} C_DIS
LIN {X -0.245,Y -478.396,Z 339.214,A 0.000,B 0.000,C 90.000,E1 74.574} C_DIS
LIN {X -0.189,Y -480.137,Z 339.212,A 0.000,B 0.000,C 90.000,E1 74.102} C_DIS
LIN {X 0.010,Y -482.181,Z 339.209,A 0.000,B 0.000,C 90.000,E1 73.614} C_DIS
LIN {X 0.175,Y -486.831,Z 339.202,A 0.000,B 0.000,C 90.000,E1 72.362} C_DIS
LIN {X 0.065,Y -490.009,Z 339.197,A 0.000,B 0.000,C 90.000,E1 71.456} C_DIS
LIN {X -0.012,Y -492.937,Z 339.192,A 0.000,B 0.000,C 90.000,E1 70.550} C_DIS
LIN {X 0.040,Y -497.605,Z 339.184,A 0.000,B 0.000,C 90.000,E1 69.028} C_DIS
LIN {X -0.105,Y -502.162,Z 339.175,A 0.000,B 0.000,C 90.000,E1 67.539} C_DIS
LIN {X -0.078,Y -507.353,Z 339.165,A 0.000,B 0.000,C 90.000,E1 65.741} C_DIS
LIN {X 0.157,Y -511.625,Z 339.157,A 0.000,B 0.000,C 90.000,E1 64.229} C_DIS
LIN {X -0.104,Y -516.662,Z 339.147,A 0.000,B 0.000,C 90.000,E1 62.487} C_DIS
LIN {X 0.072,Y -520.885,Z 339.139,A 0.000,B 0.000,C 90.000,E1 61.001} C_DIS
LIN {X 0.125,Y -525.018,Z 339.131,A 0.000,B 0.000,C 90.000,E1 59.537} C_DIS
LIN {X -0.192,Y -529.142,Z 339.123,A 0.000,B 0.000,C 90.000,E1 58.122} C_DIS
LIN {X 0.297,Y -533.165,Z 339.115,A 0.000,B 0.000,C 90.000,E1 56.628} C_DIS
LIN {X -0.024,Y -537.032,Z 339.107,A 0.000,B 0.000,C 90.000,E1 55.229} C_DIS
LIN {X 0.141,Y -540.035,Z 339.101,A 0.000,B 0.000,C 90.000,E1 54.069} C_DIS
LIN {X 0.223,Y -542.807,Z 339.094,A 0.000,B 0.000,C 90.000,E1 52.924} C_DIS
LIN {X -0.050,Y -545.966,Z 339.086,A 0.000,B 0.000,C 90.000,E1 51.537} C_DIS
LIN {X 0.082,Y -548.764,Z 339.079,A 0.000,B 0.000,C 90.000,E1 50.114} C_DIS
LIN {X -0.147,Y -550.668,Z 339.072,A 0.000,B 0.000,C 90.000,E1 49.013} C_DIS
LIN {X 0.004,Y -552.358,Z 339.066,A 0.000,B 0.000,C 90.000,E1 47.877} C_DIS
LIN {X 0.121,Y -553.367,Z 339.061,A 0.000,B 0.000,C 90.000,E1 47.025} C_DIS
LIN {X -0.154,Y -554.154,Z 339.057,A 0.000,B 0.000,C 90.000,E1 46.215} C_DIS
LIN {X -0.021,Y -554.688,Z 339.052,A 0.000,B 0.000,C 90.000,E1 45.364} C_DIS
LIN {X -0.233,Y -554.958,Z 339.046,A 0.000,B 0.000,C 90.000,E1 44.271} C_DIS
LIN {X -0.142,Y -554.956,Z 339.043,A 0.000,B 0.000,C 90.000,E1 43.704} C_DIS
LIN {X 0.007,Y -554.814,Z 339.038,A 0.000,B 0.000,C 90.000,E1 42.852} C_DIS
LIN {X 0.155,Y -554.484,Z 339.033,A 0.000,B 0.000,C 90.000,E1 42.000} C_DIS
LIN {X 0.007,Y -553.472,Z 339.026,A 0.000,B 0.000,C 90.000,E1 40.620} C_DIS
LIN {X 0.258,Y -552.090,Z 339.018,A 0.000,B 0.000,C 90.000,E1 39.197} C_DIS
LIN {X 0.074,Y -550.768,Z 339.012,A 0.000,B 0.000,C 90.000,E1 38.096} C_DIS
LIN {X 0.026,Y -548.405,Z 339.001,A 0.000,B 0.000,C 90.000,E1 36.137} C_DIS
LIN {X -0.014,Y -546.325,Z 338.991,A 0.000,B 0.000,C 90.000,E1 34.452} C_DIS
LIN {X -0.185,Y -543.699,Z 338.979,A 0.000,B 0.000,C 90.000,E1 32.212} C_DIS
LIN {X 0.290,Y -541.841,Z 338.969,A 0.000,B 0.000,C 90.000,E1 30.463} C_DIS
LIN {X 0.178,Y -539.932,Z 338.958,A 0.000,B 0.000,C 90.000,E1 28.487} C_DIS
LIN {X 0.025,Y -538.188,Z 338.949,A 0.000,B 0.000,C 90.000,E1 26.796} C_DIS
LIN {X 0.280,Y -536.292,Z 338.938,A 0.000,B 0.000,C 90.000,E1 24.771} C_DIS
LIN {X 0.065,Y -534.789,Z 338.928,A 0.000,B 0.000,C 90.000,E1 23.078} C_DIS
LIN {X -0.189,Y -533.255,Z 338.917,A 0.000,B 0.000,C 90.000,E1 21.099} C_DIS
LIN {X -0.171,Y -532.093,Z 338.906,A 0.000,B 0.000,C 90.000,E1 19.087} C_DIS
LIN {X -0.151,Y -530.838,Z 338.892,A 0.000,B 0.000,C 90.000,E1 16.496} C_DIS
LIN {X 0.035,Y -529.995,Z 338.877,A 0.000,B 0.000,C 90.000,E1 13.883} C_DIS
LIN {X -0.094,Y -529.768,Z 338.864,A 0.000,B 0.000,C 90.000,E1 11.591} C_DIS
LIN {X 0.085,Y -530.111,Z 338.852,A 0.000,B 0.000,C 90.000,E1 9.265} C_DIS
LIN {X 0.161,Y -530.952,Z 338.837,A 0.000,B 0.000,C 90.000,E1 6.663} C_DIS
LIN {X 0.192,Y -531.703,Z 338.829,A 0.000,B 0.000,C 90.000,E1 5.220} C_DIS
LIN {X 0.166,Y -534.213,Z 338.810,A 0.000,B 0.000,C 90.000,E1 1.776} C_DIS
LIN {X 0.212,Y -536.706,Z 338.796,A 0.000,B 0.000,C 90.000,E1 359.198} C_DIS
LIN {X -0.197,Y -539.977,Z 338.781,A 0.000,B 0.000,C 90.000,E1 356.674} C_DIS
LIN {X -0.118,Y -541.211,Z 338.777,A 0.000,B 0.000,C 90.000,E1 355.812} C_DIS
LIN {X 0.054,Y -543.085,Z 338.769,A 0.000,B 0.000,C 90.000,E1 354.375} C_DIS
LIN {X 0.158,Y -544.258,Z 338.764,A 0.000,B 0.000,C 90.000,E1 353.514} C_DIS
LIN {X -0.243,Y -549.824,Z 338.748,A 0.000,B 0.000,C 90.000,E1 350.735} C_DIS
LIN {X 0.033,Y -554.704,Z 338.736,A 0.000,B 0.000,C 90.000,E1 348.465} C_DIS
LIN {X -0.248,Y -561.703,Z 338.722,A 0.000,B 0.000,C 90.000,E1 345.992} C_DIS
LIN {X 0.212,Y -568.109,Z 338.710,A 0.000,B 0.000,C 90.000,E1 343.740} C_DIS
LIN {X -0.244,Y -572.442,Z 338.702,A 0.000,B 0.000,C 90.000,E1 342.417} C_DIS
LIN {X -0.082,Y -575.012,Z 338.698,A 0.000,B 0.000,C 90.000,E1 341.583} C_DIS
LIN {X -0.240,Y -579.358,Z 338.690,A 0.000,B 0.000,C 90.000,E1 340.242} C_DIS
LIN {X 0.083,Y -584.481,Z 338.681,A 0.000,B 0.000,C 90.000,E1 338.592} C_DIS
LIN {X 0.190,Y -589.687,Z 338.672,A 0.000,B 0.000,C 90.000,E1 336.975} C_DIS
LIN {X 0.225,Y -596.857,Z 338.660,A 0.000,B 0.000,C 90.000,E1 334.845} C_DIS
LIN {X -0.172,Y -601.467,Z 338.653,A 0.000,B 0.000,C 90.000,E1 333.563} C_DIS
LIN {X 0.102,Y -605.141,Z 338.647,A 0.000,B 0.000,C 90.000,E1 332.487} C_DIS
LIN {X 0.121,Y -609.785,Z 338.640,A 0.000,B 0.000,C 90.000,E1 331.179} C_DIS
LIN {X -0.087,Y -617.379,Z 338.628,A 0.000,B 0.000,C 90.000,E1 329.125} C_DIS
LIN {X -0.071,Y -622.010,Z 338.621,A 0.000,B 0.000,C 90.000,E1 327.837} C_DIS
LIN {X 0.025,Y -626.438,Z 338.614,A 0.000,B 0.000,C 90.000,E1 326.548} C_DIS
LIN {X -0.164,Y -628.923,Z 338.610,A 0.000,B 0.000,C 90.000,E1 325.801} C_DIS
LIN {X -0.126,Y -633.641,Z 338.602,A 0.000,B 0.000,C 90.000,E1 324.276} C_DIS
LIN {X -0.138,Y -638.102,Z 338.593,A 0.000,B 0.000,C 90.000,E1 322.763} C_DIS
LIN {X -0.155,Y -643.124,Z 338.583,A 0.000,B 0.000,C 90.000,E1 321.009} C_DIS
LIN {X -0.067,Y -648.356,Z 338.574,A 0.000,B 0.000,C 90.000,E1 319.256} C_DIS
LIN {X 0.062,Y -652.816,Z 338.565,A 0.000,B 0.000,C 90.000,E1 317.757} C_DIS
LIN {X -0.243,Y -659.901,Z 338.553,A 0.000,B 0.000,C 90.000,E1 315.567} C_DIS
LIN {X -0.335,Y -663.745,Z 338.546,A 0.000,B 0.000,C 90.000,E1 314.352} C_DIS
LIN {X 0.115,Y -667.498,Z 338.540,A 0.000,B 0.000,C 90.000,E1 313.095} C_DIS
LIN {X -0.309,Y -671.861,Z 338.531,A 0.000,B 0.000,C 90.000,E1 311.676} C_DIS
LIN {X -0.179,Y -675.180,Z 338.525,A 0.000,B 0.000,C 90.000,E1 310.458} C_DIS
LIN {X -0.022,Y -677.683,Z 338.519,A 0.000,B 0.000,C 90.000,E1 309.483} C_DIS
LIN {X -0.238,Y -680.670,Z 338.513,A 0.000,B 0.000,C 90.000,E1 308.302} C_DIS
LIN {X -0.257,Y -683.731,Z 338.505,A 0.000,B 0.000,C 90.000,E1 306.870} C_DIS
LIN {X -0.220,Y -686.167,Z 338.497,A 0.000,B 0.000,C 90.000,E1 305.438} C_DIS
LIN {X -0.193,Y -687.295,Z 338.492,A 0.000,B 0.000,C 90.000,E1 304.485} C_DIS
LIN {X -0.344,Y -687.964,Z 338.488,A 0.000,B 0.000,C 90.000,E1 303.785} C_DIS
LIN {X -0.126,Y -688.325,Z 338.485,A 0.000,B 0.000,C 90.000,E1 303.293} C_DIS
LIN {X 0.302,Y -688.511,Z 338.481,A 0.000,B 0.000,C 90.000,E1 302.546} C_DIS
LIN {X -0.215,Y -688.411,Z 338.477,A 0.000,B 0.000,C 90.000,E1 301.878} C_DIS
LIN {X 0.215,Y -688.066,Z 338.473,A 0.000,B 0.000,C 90.000,E1 301.131} C_DIS
LIN {X -0.305,Y -687.448,Z 338.469,A 0.000,B 0.000,C 90.000,E1 300.463} C_DIS
LIN {X -0.235,Y -686.648,Z 338.465,A 0.000,B 0.000,C 90.000,E1 299.745} C_DIS
LIN {X 0.381,Y -685.089,Z 338.460,A 0.000,B 0.000,C 90.000,E1 298.743} C_DIS
LIN {X 0.105,Y -683.734,Z 338.456,A 0.000,B 0.000,C 90.000,E1 298.052} C_DIS
LIN {X -0.253,Y -681.706,Z 338.451,A 0.000,B 0.000,C 90.000,E1 297.129} C_DIS
LIN {X -0.041,Y -679.550,Z 338.445,A 0.000,B 0.000,C 90.000,E1 296.155} C_DIS
LIN {X -0.160,Y -677.214,Z 338.440,A 0.000,B 0.000,C 90.000,E1 295.207} C_DIS
LIN {X -0.221,Y -673.483,Z 338.432,A 0.000,B 0.000,C 90.000,E1 293.770} C_DIS
LIN {X 0.033,Y -671.563,Z 338.428,A 0.000,B 0.000,C 90.000,E1 293.025} C_DIS
LIN {X -0.138,Y -667.498,Z 338.420,A 0.000,B 0.000,C 90.000,E1 291.589} C_DIS
LIN {X 0.004,Y -662.295,Z 338.409,A 0.000,B 0.000,C 90.000,E1 289.631} C_DIS
LIN {X -0.197,Y -658.590,Z 338.401,A 0.000,B 0.000,C 90.000,E1 288.181} C_DIS
LIN {X -0.134,Y -652.868,Z 338.387,A 0.000,B 0.000,C 90.000,E1 285.717} C_DIS
LIN {X -0.279,Y -647.323,Z 338.372,A 0.000,B 0.000,C 90.000,E1 283.008} C_DIS
LIN {X -0.271,Y -642.526,Z 338.356,A 0.000,B 0.000,C 90.000,E1 280.018} C_DIS
LIN {X 0.026,Y -638.739,Z 338.336,A 0.000,B 0.000,C 90.000,E1 276.486} C_DIS
LIN {X -0.199,Y -637.230,Z 338.324,A 0.000,B 0.000,C 90.000,E1 274.245} C_DIS
LIN {X -0.085,Y -636.316,Z 338.310,A 0.000,B 0.000,C 90.000,E1 271.718} C_DIS
LIN {X -0.311,Y -636.225,Z 338.294,A 0.000,B 0.000,C 90.000,E1 268.969} C_DIS
LIN {X 0.012,Y -636.909,Z 338.282,A 0.000,B 0.000,C 90.000,E1 266.674} C_DIS
LIN {X 0.229,Y -637.813,Z 338.272,A 0.000,B 0.000,C 90.000,E1 264.894} C_DIS
LIN {X -0.120,Y -638.859,Z 338.262,A 0.000,B 0.000,C 90.000,E1 263.166} C_DIS
LIN {X 0.262,Y -640.137,Z 338.252,A 0.000,B 0.000,C 90.000,E1 261.376} C_DIS
LIN {X -0.056,Y -641.178,Z 338.245,A 0.000,B 0.000,C 90.000,E1 260.151} C_DIS
LIN {X 0.177,Y -644.589,Z 338.227,A 0.000,B 0.000,C 90.000,E1 256.881} C_DIS
LIN {X 0.070,Y -646.046,Z 338.220,A 0.000,B 0.000,C 90.000,E1 255.644} C_DIS
LIN {X -0.218,Y -646.578,Z 338.218,A 0.000,B 0.000,C 90.000,E1 255.172} C_DIS
LIN {X 0.149,Y -647.053,Z 338.213,A 0.000,B 0.000,C 90.000,E1 254.393} C_DIS
LIN {X -0.232,Y -647.573,Z 338.208,A 0.000,B 0.000,C 90.000,E1 253.433} C_DIS
LIN {X -0.037,Y -647.670,Z 338.204,A 0.000,B 0.000,C 90.000,E1 252.670} C_DIS
LIN {X -0.215,Y -647.530,Z 338.198,A 0.000,B 0.000,C 90.000,E1 251.692} C_DIS
LIN {X 0.106,Y -647.296,Z 338.195,A 0.000,B 0.000,C 90.000,E1 251.167} C_DIS
LIN {X -0.072,Y -646.430,Z 338.190,A 0.000,B 0.000,C 90.000,E1 250.188} C_DIS
LIN {X -0.257,Y -644.938,Z 338.184,A 0.000,B 0.000,C 90.000,E1 249.209} C_DIS
LIN {X -0.357,Y -644.063,Z 338.182,A 0.000,B 0.000,C 90.000,E1 248.720} C_DIS
LIN {X 0.197,Y -642.481,Z 338.177,A 0.000,B 0.000,C 90.000,E1 247.922} C_DIS
LIN {X 0.196,Y -640.053,Z 338.172,A 0.000,B 0.000,C 90.000,E1 246.922} C_DIS
LIN {X 0.169,Y -637.263,Z 338.166,A 0.000,B 0.000,C 90.000,E1 245.921} C_DIS
LIN {X 0.056,Y -635.050,Z 338.162,A 0.000,B 0.000,C 90.000,E1 245.177} C_DIS
LIN {X 0.186,Y -632.624,Z 338.158,A 0.000,B 0.000,C 90.000,E1 244.409} C_DIS
LIN {X 0.324,Y -629.117,Z 338.152,A 0.000,B 0.000,C 90.000,E1 243.384} C_DIS
LIN {X -0.159,Y -626.370,Z 338.148,A 0.000,B 0.000,C 90.000,E1 242.666} C_DIS
LIN {X 0.196,Y -619.003,Z 338.137,A 0.000,B 0.000,C 90.000,E1 240.589} C_DIS
LIN {X -0.380,Y -616.288,Z 338.132,A 0.000,B 0.000,C 90.000,E1 239.871} C_DIS
LIN {X 0.061,Y -610.639,Z 338.124,A 0.000,B 0.000,C 90.000,E1 238.280} C_DIS
LIN {X -0.078,Y -605.910,Z 338.117,A 0.000,B 0.000,C 90.000,E1 236.993} C_DIS
LIN {X -0.133,Y -603.028,Z 338.112,A 0.000,B 0.000,C 90.000,E1 236.215} C_DIS
LIN {X -0.079,Y -593.711,Z 338.098,A 0.000,B 0.000,C 90.000,E1 233.577} C_DIS
LIN {X 0.105,Y -590.885,Z 338.093,A 0.000,B 0.000,C 90.000,E1 232.763} C_DIS
LIN {X 0.220,Y -584.029,Z 338.083,A 0.000,B 0.000,C 90.000,E1 230.884} C_DIS
LIN {X -0.337,Y -574.798,Z 338.068,A 0.000,B 0.000,C 90.000,E1 228.243} C_DIS
LIN {X -0.048,Y -569.429,Z 338.059,A 0.000,B 0.000,C 90.000,E1 226.581} C_DIS
LIN {X 0.288,Y -562.166,Z 338.047,A 0.000,B 0.000,C 90.000,E1 224.352} C_DIS
LIN {X 0.302,Y -556.728,Z 338.037,A 0.000,B 0.000,C 90.000,E1 222.690} C_DIS
LIN {X 0.119,Y -553.188,Z 338.031,A 0.000,B 0.000,C 90.000,E1 221.595} C_DIS
LIN {X 0.072,Y -546.101,Z 338.019,A 0.000,B 0.000,C 90.000,E1 219.358} C_DIS
LIN {X 0.172,Y -541.805,Z 338.011,A 0.000,B 0.000,C 90.000,E1 217.935} C_DIS
LIN {X 0.001,Y -534.336,Z 337.997,A 0.000,B 0.000,C 90.000,E1 215.391} C_DIS
LIN {X -0.289,Y -526.603,Z 337.981,A 0.000,B 0.000,C 90.000,E1 212.546} C_DIS
LIN {X -0.139,Y -521.038,Z 337.968,A 0.000,B 0.000,C 90.000,E1 210.207} C_DIS
LIN {X 0.013,Y -517.011,Z 337.958,A 0.000,B 0.000,C 90.000,E1 208.437} C_DIS
LIN {X 0.065,Y -513.147,Z 337.948,A 0.000,B 0.000,C 90.000,E1 206.668} C_DIS
LIN {X 0.129,Y -508.662,Z 337.937,A 0.000,B 0.000,C 90.000,E1 204.591} C_DIS
LIN {X 0.080,Y -504.049,Z 337.925,A 0.000,B 0.000,C 90.000,E1 202.514} C_DIS
LIN {X -0.160,Y -500.697,Z 337.917,A 0.000,B 0.000,C 90.000,E1 201.046} C_DIS
LIN {X 0.076,Y -496.614,Z 337.907,A 0.000,B 0.000,C 90.000,E1 199.214} C_DIS
LIN {X -0.022,Y -491.416,Z 337.893,A 0.000,B 0.000,C 90.000,E1 196.804} C_DIS
LIN {X -0.190,Y -488.354,Z 337.885,A 0.000,B 0.000,C 90.000,E1 195.300} C_DIS
LIN {X 0.003,Y -483.693,Z 337.871,A 0.000,B 0.000,C 90.000,E1 192.827} C_DIS
LIN {X 0.239,Y -480.332,Z 337.861,A 0.000,B 0.000,C 90.000,E1 190.950} C_DIS
LIN {X -0.100,Y -477.578,Z 337.852,A 0.000,B 0.000,C 90.000,E1 189.443} C_DIS
LIN {X -0.038,Y -473.427,Z 337.839,A 0.000,B 0.000,C 90.000,E1 186.947} C_DIS
LIN {X -0.044,Y -469.199,Z 337.823,A 0.000,B 0.000,C 90.000,E1 184.131} C_DIS
LIN {X 0.014,Y -466.791,Z 337.812,A 0.000,B 0.000,C 90.000,E1 182.236} C_DIS
LIN {X 0.161,Y -463.211,Z 337.793,A 0.000,B 0.000,C 90.000,E1 178.740} C_DIS
LIN {X -0.027,Y -460.725,Z 337.772,A 0.000,B 0.000,C 90.000,E1 174.951} C_DIS
LIN {X 0.112,Y -460.020,Z 337.749,A 0.000,B 0.000,C 90.000,E1 170.792} C_DIS
LIN {X 0.150,Y -460.635,Z 337.726,A 0.000,B 0.000,C 90.000,E1 166.645} C_DIS
LIN {X 0.179,Y -462.527,Z 337.707,A 0.000,B 0.000,C 90.000,E1 163.142} C_DIS
LIN {X -0.243,Y -466.020,Z 337.685,A 0.000,B 0.000,C 90.000,E1 159.390} C_DIS
LIN {X -0.220,Y -470.655,Z 337.666,A 0.000,B 0.000,C 90.000,E1 155.921} C_DIS
LIN {X -0.119,Y -477.992,Z 337.644,A 0.000,B 0.000,C 90.000,E1 151.847} C_DIS
LIN {X 0.262,Y -487.453,Z 337.621,A 0.000,B 0.000,C 90.000,E1 147.788} C_DIS
LIN {X 0.025,Y -496.180,Z 337.604,A 0.000,B 0.000,C 90.000,E1 144.769} C_DIS
LIN {X -0.070,Y -501.600,Z 337.594,A 0.000,B 0.000,C 90.000,E1 142.970} C_DIS
LIN {X 0.175,Y -505.186,Z 337.588,A 0.000,B 0.000,C 90.000,E1 141.743} C_DIS
LIN {X 0.076,Y -508.552,Z 337.581,A 0.000,B 0.000,C 90.000,E1 140.561} C_DIS
LIN {X 0.116,Y -510.880,Z 337.576,A 0.000,B 0.000,C 90.000,E1 139.666} C_DIS
LIN {X 0.346,Y -514.488,Z 337.568,A 0.000,B 0.000,C 90.000,E1 138.162} C_DIS
LIN {X 0.061,Y -516.261,Z 337.563,A 0.000,B 0.000,C 90.000,E1 137.310} C_DIS
LIN {X -0.128,Y -517.270,Z 337.560,A 0.000,B 0.000,C 90.000,E1 136.743} C_DIS
LIN {X -0.105,Y -518.800,Z 337.553,A 0.000,B 0.000,C 90.000,E1 135.567} C_DIS
LIN {X 0.301,Y -519.817,Z 337.547,A 0.000,B 0.000,C 90.000,E1 134.352} C_DIS
LIN {X 0.070,Y -520.155,Z 337.542,A 0.000,B 0.000,C 90.000,E1 133.500} C_DIS
LIN {X -0.247,Y -520.272,Z 337.535,A 0.000,B 0.000,C 90.000,E1 132.366} C_DIS
LIN {X -0.024,Y -520.029,Z 337.532,A 0.000,B 0.000,C 90.000,E1 131.757} C_DIS
LIN {X 0.199,Y -519.729,Z 337.529,A 0.000,B 0.000,C 90.000,E1 131.148} C_DIS
LIN {X -0.097,Y -518.570,Z 337.522,A 0.000,B 0.000,C 90.000,E1 130.011} C_DIS
LIN {X 0.051,Y -517.514,Z 337.517,A 0.000,B 0.000,C 90.000,E1 129.116} C_DIS
LIN {X 0.050,Y -515.524,Z 337.509,A 0.000,B 0.000,C 90.000,E1 127.649} C_DIS
LIN {X 0.112,Y -513.487,Z 337.501,A 0.000,B 0.000,C 90.000,E1 126.171} C_DIS
LIN {X -0.194,Y -511.637,Z 337.495,A 0.000,B 0.000,C 90.000,E1 125.025} C_DIS
LIN {X -0.027,Y -510.189,Z 337.490,A 0.000,B 0.000,C 90.000,E1 124.119} C_DIS
LIN {X 0.074,Y -507.414,Z 337.481,A 0.000,B 0.000,C 90.000,E1 122.625} C_DIS
LIN {X 0.004,Y -503.685,Z 337.471,A 0.000,B 0.000,C 90.000,E1 120.846} C_DIS
LIN {X 0.149,Y -500.456,Z 337.463,A 0.000,B 0.000,C 90.000,E1 119.333} C_DIS
LIN {X -0.049,Y -497.803,Z 337.456,A 0.000,B 0.000,C 90.000,E1 118.153} C_DIS
LIN {X -0.209,Y -493.647,Z 337.446,A 0.000,B 0.000,C 90.000,E1 116.360} C_DIS
LIN {X -0.048,Y -490.072,Z 337.438,A 0.000,B 0.000,C 90.000,E1 114.823} C_DIS
LIN {X 0.062,Y -487.080,Z 337.431,A 0.000,B 0.000,C 90.000,E1 113.590} C_DIS
LIN {X -0.122,Y -483.965,Z 337.424,A 0.000,B 0.000,C 90.000,E1 112.386} C_DIS
LIN {X -0.105,Y -482.458,Z 337.421,A 0.000,B 0.000,C 90.000,E1 111.770} C_DIS
LIN {X -0.282,Y -478.301,Z 337.412,A 0.000,B 0.000,C 90.000,E1 110.248} C_DIS
LIN {X 0.099,Y -474.708,Z 337.405,A 0.000,B 0.000,C 90.000,E1 108.960} C_DIS
LIN {X 0.075,Y -470.017,Z 337.397,A 0.000,B 0.000,C 90.000,E1 107.402} C_DIS
LIN {X 0.163,Y -466.075,Z 337.390,A 0.000,B 0.000,C 90.000,E1 106.134} C_DIS
LIN {X 0.119,Y -465.292,Z 337.388,A 0.000,B 0.000,C 90.000,E1 105.898} C_DIS
LIN {X 0.078,Y -465.298,Z 337.388,A 0.000,B 0.000,C 90.000,E1 105.898} C_DIS
LIN {X -0.060,Y -467.787,Z 337.383,A 0.000,B 0.000,C 90.000,E1 104.898} C_DIS
LIN {X -0.088,Y -475.992,Z 337.357,A 0.000,B 0.000,C 90.000,E1 100.197} C_DIS
LIN {X 0.060,Y -476.690,Z 337.353,A 0.000,B 0.000,C 90.000,E1 99.557} C_DIS
LIN {X 0.186,Y -481.933,Z 337.331,A 0.000,B 0.000,C 90.000,E1 95.511} C_DIS
LIN {X 0.034,Y -482.207,Z 337.329,A 0.000,B 0.000,C 90.000,E1 95.220} C_DIS
LIN {X -0.028,Y -485.403,Z 337.305,A 0.000,B 0.000,C 90.000,E1 90.917} C_DIS
LIN {X -0.203,Y -485.528,Z 337.303,A 0.000,B 0.000,C 90.000,E1 90.630} C_DIS
LIN {X 0.004,Y -486.364,Z 337.281,A 0.000,B 0.000,C 90.000,E1 86.617} C_DIS
LIN {X -0.171,Y -486.367,Z 337.280,A 0.000,B 0.000,C 90.000,E1 86.331} C_DIS
LIN {X 0.163,Y -485.675,Z 337.273,A 0.000,B 0.000,C 90.000,E1 85.065} C_DIS
LIN {X -0.147,Y -484.692,Z 337.254,A 0.000,B 0.000,C 90.000,E1 81.724} C_DIS
LIN {X 0.199,Y -484.491,Z 337.252,A 0.000,B 0.000,C 90.000,E1 81.376} C_DIS
LIN {X -0.266,Y -480.664,Z 337.228,A 0.000,B 0.000,C 90.000,E1 77.117} C_DIS
LIN {X 0.169,Y -480.418,Z 337.227,A 0.000,B 0.000,C 90.000,E1 76.756} C_DIS
LIN {X 0.180,Y -477.409,Z 337.216,A 0.000,B 0.000,C 90.000,E1 74.810} C_DIS
LIN {X 0.139,Y -477.414,Z 337.216,A 0.000,B 0.000,C 90.000,E1 74.810} C_DIS
LIN {X 0.130,Y -479.453,Z 337.213,A 0.000,B 0.000,C 90.000,E1 74.283} C_DIS
LIN {X -0.137,Y -481.129,Z 337.210,A 0.000,B 0.000,C 90.000,E1 73.850} C_DIS
LIN {X -0.051,Y -481.824,Z 337.209,A 0.000,B 0.000,C 90.000,E1 73.685} C_DIS
LIN {X 0.244,Y -486.217,Z 337.203,A 0.000,B 0.000,C 90.000,E1 72.417} C_DIS
LIN {X 0.130,Y -489.341,Z 337.197,A 0.000,B 0.000,C 90.000,E1 71.511} C_DIS
LIN {X -0.082,Y -493.125,Z 337.191,A 0.000,B 0.000,C 90.000,E1 70.315} C_DIS
LIN {X 0.146,Y -497.716,Z 337.182,A 0.000,B 0.000,C 90.000,E1 68.773} C_DIS
LIN {X -0.064,Y -501.326,Z 337.176,A 0.000,B 0.000,C 90.000,E1 67.592} C_DIS
LIN {X -0.049,Y -506.490,Z 337.166,A 0.000,B 0.000,C 90.000,E1 65.793} C_DIS
LIN {X 0.176,Y -510.771,Z 337.157,A 0.000,B 0.000,C 90.000,E1 64.280} C_DIS
LIN {X 0.013,Y -514.954,Z 337.149,A 0.000,B 0.000,C 90.000,E1 62.820} C_DIS
LIN {X -0.301,Y -519.210,Z 337.141,A 0.000,B 0.000,C 90.000,E1 61.385} C_DIS
LIN {X 0.175,Y -523.373,Z 337.133,A 0.000,B 0.000,C 90.000,E1 59.871} C_DIS
LIN {X 0.238,Y -528.341,Z 337.123,A 0.000,B 0.000,C 90.000,E1 58.122} C_DIS
LIN {X -0.021,Y -532.405,Z 337.115,A 0.000,B 0.000,C 90.000,E1 56.707} C_DIS
LIN {X 0.078,Y -536.300,Z 337.107,A 0.000,B 0.000,C 90.000,E1 55.261} C_DIS
LIN {X 0.103,Y -539.318,Z 337.101,A 0.000,B 0.000,C 90.000,E1 54.116} C_DIS
LIN {X -0.145,Y -542.121,Z 337.094,A 0.000,B 0.000,C 90.000,E1 53.004} C_DIS
LIN {X 0.333,Y -545.307,Z 337.087,A 0.000,B 0.000,C 90.000,E1 51.537} C_DIS
LIN {X 0.102,Y -548.134,Z 337.079,A 0.000,B 0.000,C 90.000,E1 50.150} C_DIS
LIN {X 0.171,Y -549.655,Z 337.074,A 0.000,B 0.000,C 90.000,E1 49.299} C_DIS
LIN {X 0.312,Y -551.384,Z 337.068,A 0.000,B 0.000,C 90.000,E1 48.162} C_DIS
LIN {X 0.068,Y -552.888,Z 337.062,A 0.000,B 0.000,C 90.000,E1 47.067} C_DIS
LIN {X 0.192,Y -553.739,Z 337.057,A 0.000,B 0.000,C 90.000,E1 46.215} C_DIS
LIN {X -0.073,Y -554.362,Z 337.052,A 0.000,B 0.000,C 90.000,E1 45.405} C_DIS
LIN {X 0.058,Y -554.747,Z 337.048,A 0.000,B 0.000,C 90.000,E1 44.555} C_DIS
LIN {X 0.196,Y -554.924,Z 337.043,A 0.000,B 0.000,C 90.000,E1 43.704} C_DIS
LIN {X -0.004,Y -554.790,Z 337.037,A 0.000,B 0.000,C 90.000,E1 42.609} C_DIS
LIN {X 0.143,Y -554.515,Z 337.032,A 0.000,B 0.000,C 90.000,E1 41.757} C_DIS
LIN {X -0.071,Y -553.807,Z 337.026,A 0.000,B 0.000,C 90.000,E1 40.663} C_DIS
LIN {X -0.237,Y -552.808,Z 337.020,A 0.000,B 0.000,C 90.000,E1 39.564} C_DIS
LIN {X -0.347,Y -551.323,Z 337.012,A 0.000,B 0.000,C 90.000,E1 38.177} C_DIS
LIN {X 0.012,Y -549.329,Z 337.003,A 0.000,B 0.000,C 90.000,E1 36.457} C_DIS
LIN {X 0.007,Y -547.287,Z 336.993,A 0.000,B 0.000,C 90.000,E1 34.771} C_DIS
LIN {X -0.282,Y -544.638,Z 336.981,A 0.000,B 0.000,C 90.000,E1 32.546} C_DIS
LIN {X 0.214,Y -542.770,Z 336.971,A 0.000,B 0.000,C 90.000,E1 30.797} C_DIS
LIN {X -0.135,Y -540.579,Z 336.959,A 0.000,B 0.000,C 90.000,E1 28.565} C_DIS
LIN {X 0.001,Y -539.154,Z 336.951,A 0.000,B 0.000,C 90.000,E1 27.129} C_DIS
LIN {X -0.198,Y -537.232,Z 336.940,A 0.000,B 0.000,C 90.000,E1 25.155} C_DIS
LIN {X 0.033,Y -535.460,Z 336.929,A 0.000,B 0.000,C 90.000,E1 23.131} C_DIS
LIN {X 0.288,Y -533.928,Z 336.917,A 0.000,B 0.000,C 90.000,E1 21.099} C_DIS
LIN {X -0.181,Y -532.768,Z 336.906,A 0.000,B 0.000,C 90.000,E1 19.141} C_DIS
LIN {X -0.116,Y -531.389,Z 336.890,A 0.000,B 0.000,C 90.000,E1 16.260} C_DIS
LIN {X 0.090,Y -530.580,Z 336.876,A 0.000,B 0.000,C 90.000,E1 13.647} C_DIS
LIN {X -0.129,Y -530.407,Z 336.863,A 0.000,B 0.000,C 90.000,E1 11.366} C_DIS
LIN {X 0.133,Y -530.737,Z 336.852,A 0.000,B 0.000,C 90.000,E1 9.321} C_DIS
LIN {X 0.226,Y -531.549,Z 336.838,A 0.000,B 0.000,C 90.000,E1 6.720} C_DIS
LIN {X 0.266,Y -532.291,Z 336.830,A 0.000,B 0.000,C 90.000,E1 5.277} C_DIS
LIN {X 0.247,Y -534.763,Z 336.810,A 0.000,B 0.000,C 90.000,E1 1.835} C_DIS
LIN {X 0.217,Y -537.253,Z 336.796,A 0.000,B 0.000,C 90.000,E1 359.198} C_DIS
LIN {X -0.175,Y -540.484,Z 336.781,A 0.000,B 0.000,C 90.000,E1 356.674} C_DIS
LIN {X -0.074,Y -542.010,Z 336.775,A 0.000,B 0.000,C 90.000,E1 355.527} C_DIS
LIN {X 0.090,Y -543.458,Z 336.769,A 0.000,B 0.000,C 90.000,E1 354.375} C_DIS
LIN {X 0.198,Y -544.568,Z 336.764,A 0.000,B 0.000,C 90.000,E1 353.514} C_DIS
LIN {X -0.193,Y -550.069,Z 336.748,A 0.000,B 0.000,C 90.000,E1 350.735} C_DIS
LIN {X -0.274,Y -552.899,Z 336.741,A 0.000,B 0.000,C 90.000,E1 349.342} C_DIS
LIN {X -0.200,Y -556.337,Z 336.733,A 0.000,B 0.000,C 90.000,E1 347.937} C_DIS
LIN {X -0.187,Y -561.816,Z 336.722,A 0.000,B 0.000,C 90.000,E1 345.992} C_DIS
LIN {X 0.181,Y -565.744,Z 336.714,A 0.000,B 0.000,C 90.000,E1 344.574} C_DIS
LIN {X -0.177,Y -572.520,Z 336.702,A 0.000,B 0.000,C 90.000,E1 342.417} C_DIS
LIN {X -0.189,Y -577.624,Z 336.693,A 0.000,B 0.000,C 90.000,E1 340.786} C_DIS
LIN {X 0.215,Y -580.236,Z 336.689,A 0.000,B 0.000,C 90.000,E1 339.934} C_DIS
LIN {X 0.018,Y -585.347,Z 336.680,A 0.000,B 0.000,C 90.000,E1 338.337} C_DIS
LIN {X -0.086,Y -590.592,Z 336.671,A 0.000,B 0.000,C 90.000,E1 336.741} C_DIS
LIN {X 0.129,Y -598.749,Z 336.658,A 0.000,B 0.000,C 90.000,E1 334.332} C_DIS
LIN {X 0.303,Y -603.379,Z 336.650,A 0.000,B 0.000,C 90.000,E1 332.999} C_DIS
LIN {X 0.199,Y -609.888,Z 336.640,A 0.000,B 0.000,C 90.000,E1 331.179} C_DIS
LIN {X -0.032,Y -618.459,Z 336.627,A 0.000,B 0.000,C 90.000,E1 328.869} C_DIS
LIN {X -0.002,Y -623.036,Z 336.620,A 0.000,B 0.000,C 90.000,E1 327.582} C_DIS
LIN {X 0.112,Y -626.568,Z 336.614,A 0.000,B 0.000,C 90.000,E1 326.548} C_DIS
LIN {X -0.076,Y -629.003,Z 336.610,A 0.000,B 0.000,C 90.000,E1 325.801} C_DIS
LIN {X -0.036,Y -633.618,Z 336.602,A 0.000,B 0.000,C 90.000,E1 324.276} C_DIS
LIN {X 0.074,Y -637.313,Z 336.595,A 0.000,B 0.000,C 90.000,E1 323.004} C_DIS
LIN {X 0.339,Y -643.658,Z 336.582,A 0.000,B 0.000,C 90.000,E1 320.723} C_DIS
LIN {X 0.017,Y -648.129,Z 336.574,A 0.000,B 0.000,C 90.000,E1 319.256} C_DIS
LIN {X 0.140,Y -652.540,Z 336.565,A 0.000,B 0.000,C 90.000,E1 317.757} C_DIS
LIN {X -0.171,Y -659.571,Z 336.553,A 0.000,B 0.000,C 90.000,E1 315.567} C_DIS
LIN {X -0.254,Y -662.659,Z 336.548,A 0.000,B 0.000,C 90.000,E1 314.595} C_DIS
LIN {X 0.176,Y -667.129,Z 336.540,A 0.000,B 0.000,C 90.000,E1 313.095} C_DIS
LIN {X -0.262,Y -670.727,Z 336.533,A 0.000,B 0.000,C 90.000,E1 311.919} C_DIS
LIN {X 0.269,Y -672.753,Z 336.529,A 0.000,B 0.000,C 90.000,E1 311.148} C_DIS
LIN {X -0.117,Y -675.330,Z 336.523,A 0.000,B 0.000,C 90.000,E1 310.216} C_DIS
LIN {X -0.392,Y -677.768,Z 336.518,A 0.000,B 0.000,C 90.000,E1 309.277} C_DIS
LIN {X -0.204,Y -680.082,Z 336.513,A 0.000,B 0.000,C 90.000,E1 308.302} C_DIS
LIN {X 0.152,Y -682.574,Z 336.506,A 0.000,B 0.000,C 90.000,E1 307.076} C_DIS
LIN {X -0.235,Y -683.095,Z 336.505,A 0.000,B 0.000,C 90.000,E1 306.870} C_DIS
LIN {X 0.147,Y -684.668,Z 336.499,A 0.000,B 0.000,C 90.000,E1 305.884} C_DIS
LIN {X -0.211,Y -685.475,Z 336.497,A 0.000,B 0.000,C 90.000,E1 305.438} C_DIS
LIN {X -0.192,Y -686.575,Z 336.492,A 0.000,B 0.000,C 90.000,E1 304.485} C_DIS
LIN {X -0.351,Y -687.204,Z 336.488,A 0.000,B 0.000,C 90.000,E1 303.785} C_DIS
LIN {X -0.137,Y -687.548,Z 336.485,A 0.000,B 0.000,C 90.000,E1 303.293} C_DIS
LIN {X 0.283,Y -687.707,Z 336.481,A 0.000,B 0.000,C 90.000,E1 302.546} C_DIS
LIN {X 0.127,Y -687.671,Z 336.478,A 0.000,B 0.000,C 90.000,E1 302.084} C_DIS
LIN {X -0.035,Y -687.358,Z 336.474,A 0.000,B 0.000,C 90.000,E1 301.386} C_DIS
LIN {X 0.026,Y -686.795,Z 336.470,A 0.000,B 0.000,C 90.000,E1 300.669} C_DIS
LIN {X -0.286,Y -685.716,Z 336.465,A 0.000,B 0.000,C 90.000,E1 299.745} C_DIS
LIN {X 0.317,Y -684.134,Z 336.460,A 0.000,B 0.000,C 90.000,E1 298.743} C_DIS
LIN {X -0.148,Y -681.758,Z 336.453,A 0.000,B 0.000,C 90.000,E1 297.590} C_DIS
LIN {X 0.271,Y -679.081,Z 336.447,A 0.000,B 0.000,C 90.000,E1 296.360} C_DIS
LIN {X -0.271,Y -676.125,Z 336.440,A 0.000,B 0.000,C 90.000,E1 295.207} C_DIS
LIN {X 0.360,Y -672.985,Z 336.433,A 0.000,B 0.000,C 90.000,E1 293.951} C_DIS
LIN {X -0.109,Y -670.419,Z 336.428,A 0.000,B 0.000,C 90.000,E1 293.025} C_DIS
LIN {X -0.301,Y -666.311,Z 336.420,A 0.000,B 0.000,C 90.000,E1 291.589} C_DIS
LIN {X -0.083,Y -661.716,Z 336.410,A 0.000,B 0.000,C 90.000,E1 289.866} C_DIS
LIN {X 0.212,Y -657.401,Z 336.401,A 0.000,B 0.000,C 90.000,E1 288.127} C_DIS
LIN {X 0.365,Y -652.178,Z 336.389,A 0.000,B 0.000,C 90.000,E1 285.898} C_DIS
LIN {X -0.009,Y -647.509,Z 336.376,A 0.000,B 0.000,C 90.000,E1 283.703} C_DIS
LIN {X 0.183,Y -641.719,Z 336.357,A 0.000,B 0.000,C 90.000,E1 280.197} C_DIS
LIN {X 0.268,Y -637.583,Z 336.336,A 0.000,B 0.000,C 90.000,E1 276.429} C_DIS
LIN {X 0.011,Y -636.077,Z 336.323,A 0.000,B 0.000,C 90.000,E1 274.188} C_DIS
LIN {X -0.311,Y -635.265,Z 336.311,A 0.000,B 0.000,C 90.000,E1 271.949} C_DIS
LIN {X -0.056,Y -635.240,Z 336.291,A 0.000,B 0.000,C 90.000,E1 268.396} C_DIS
LIN {X 0.016,Y -636.184,Z 336.277,A 0.000,B 0.000,C 90.000,E1 265.869} C_DIS
LIN {X 0.209,Y -637.138,Z 336.267,A 0.000,B 0.000,C 90.000,E1 264.090} C_DIS
LIN {X 0.102,Y -638.179,Z 336.259,A 0.000,B 0.000,C 90.000,E1 262.591} C_DIS
LIN {X 0.112,Y -639.994,Z 336.246,A 0.000,B 0.000,C 90.000,E1 260.330} C_DIS
LIN {X 0.101,Y -641.647,Z 336.237,A 0.000,B 0.000,C 90.000,E1 258.578} C_DIS
LIN {X -0.174,Y -644.387,Z 336.224,A 0.000,B 0.000,C 90.000,E1 256.353} C_DIS
LIN {X 0.020,Y -645.557,Z 336.219,A 0.000,B 0.000,C 90.000,E1 255.338} C_DIS
LIN {X 0.068,Y -646.315,Z 336.213,A 0.000,B 0.000,C 90.000,E1 254.338} C_DIS
LIN {X 0.294,Y -646.846,Z 336.208,A 0.000,B 0.000,C 90.000,E1 253.323} C_DIS
LIN {X -0.093,Y -647.084,Z 336.202,A 0.000,B 0.000,C 90.000,E1 252.362} C_DIS
LIN {X 0.284,Y -647.025,Z 336.198,A 0.000,B 0.000,C 90.000,E1 251.583} C_DIS
LIN {X 0.194,Y -646.870,Z 336.195,A 0.000,B 0.000,C 90.000,E1 251.094} C_DIS
LIN {X 0.105,Y -646.593,Z 336.192,A 0.000,B 0.000,C 90.000,E1 250.604} C_DIS
LIN {X 0.017,Y -646.174,Z 336.190,A 0.000,B 0.000,C 90.000,E1 250.115} C_DIS
LIN {X -0.165,Y -644.856,Z 336.184,A 0.000,B 0.000,C 90.000,E1 249.135} C_DIS
LIN {X 0.167,Y -643.560,Z 336.180,A 0.000,B 0.000,C 90.000,E1 248.358} C_DIS
LIN {X 0.117,Y -642.043,Z 336.176,A 0.000,B 0.000,C 90.000,E1 247.614} C_DIS
LIN {X 0.053,Y -640.276,Z 336.172,A 0.000,B 0.000,C 90.000,E1 246.869} C_DIS
LIN {X 0.229,Y -638.253,Z 336.167,A 0.000,B 0.000,C 90.000,E1 246.102} C_DIS
LIN {X 0.178,Y -635.336,Z 336.162,A 0.000,B 0.000,C 90.000,E1 245.101} C_DIS
LIN {X 0.041,Y -632.910,Z 336.158,A 0.000,B 0.000,C 90.000,E1 244.357} C_DIS
LIN {X 0.180,Y -629.423,Z 336.152,A 0.000,B 0.000,C 90.000,E1 243.332} C_DIS
LIN {X -0.304,Y -626.696,Z 336.148,A 0.000,B 0.000,C 90.000,E1 242.615} C_DIS
LIN {X 0.057,Y -620.312,Z 336.138,A 0.000,B 0.000,C 90.000,E1 240.795} C_DIS
LIN {X -0.214,Y -616.731,Z 336.132,A 0.000,B 0.000,C 90.000,E1 239.793} C_DIS
LIN {X 0.243,Y -611.215,Z 336.124,A 0.000,B 0.000,C 90.000,E1 238.201} C_DIS
LIN {X 0.117,Y -606.598,Z 336.116,A 0.000,B 0.000,C 90.000,E1 236.914} C_DIS
LIN {X 0.069,Y -603.759,Z 336.112,A 0.000,B 0.000,C 90.000,E1 236.135} C_DIS
LIN {X -0.076,Y -595.413,Z 336.099,A 0.000,B 0.000,C 90.000,E1 233.783} C_DIS
LIN {X -0.013,Y -591.675,Z 336.093,A 0.000,B 0.000,C 90.000,E1 232.718} C_DIS
LIN {X -0.155,Y -583.900,Z 336.081,A 0.000,B 0.000,C 90.000,E1 230.598} C_DIS
LIN {X -0.076,Y -578.320,Z 336.072,A 0.000,B 0.000,C 90.000,E1 228.976} C_DIS
LIN {X 0.328,Y -572.972,Z 336.063,A 0.000,B 0.000,C 90.000,E1 227.310} C_DIS
LIN {X -0.039,Y -569.381,Z 336.057,A 0.000,B 0.000,C 90.000,E1 226.257} C_DIS
LIN {X -0.182,Y -563.040,Z 336.046,A 0.000,B 0.000,C 90.000,E1 224.352} C_DIS
LIN {X -0.036,Y -555.861,Z 336.034,A 0.000,B 0.000,C 90.000,E1 222.123} C_DIS
LIN {X -0.063,Y -549.609,Z 336.023,A 0.000,B 0.000,C 90.000,E1 220.172} C_DIS
LIN {X 0.145,Y -544.428,Z 336.014,A 0.000,B 0.000,C 90.000,E1 218.463} C_DIS
LIN {X -0.067,Y -537.643,Z 336.001,A 0.000,B 0.000,C 90.000,E1 216.217} C_DIS
LIN {X 0.097,Y -533.639,Z 335.993,A 0.000,B 0.000,C 90.000,E1 214.771} C_DIS
LIN {X 0.226,Y -526.073,Z 335.977,A 0.000,B 0.000,C 90.000,E1 211.878} C_DIS
LIN {X 0.294,Y -521.959,Z 335.968,A 0.000,B 0.000,C 90.000,E1 210.129} C_DIS
LIN {X 0.084,Y -518.607,Z 335.960,A 0.000,B 0.000,C 90.000,E1 208.693} C_DIS
LIN {X -0.171,Y -514.007,Z 335.948,A 0.000,B 0.000,C 90.000,E1 206.668} C_DIS
LIN {X -0.191,Y -510.155,Z 335.938,A 0.000,B 0.000,C 90.000,E1 204.899} C_DIS
LIN {X -0.127,Y -508.204,Z 335.933,A 0.000,B 0.000,C 90.000,E1 204.003} C_DIS
LIN {X -0.107,Y -504.906,Z 335.925,A 0.000,B 0.000,C 90.000,E1 202.514} C_DIS
LIN {X 0.317,Y -501.549,Z 335.917,A 0.000,B 0.000,C 90.000,E1 200.972} C_DIS
LIN {X 0.029,Y -498.170,Z 335.908,A 0.000,B 0.000,C 90.000,E1 199.504} C_DIS
LIN {X 0.032,Y -494.197,Z 335.898,A 0.000,B 0.000,C 90.000,E1 197.692} C_DIS
LIN {X 0.162,Y -489.904,Z 335.887,A 0.000,B 0.000,C 90.000,E1 195.552} C_DIS
LIN {X 0.055,Y -485.233,Z 335.873,A 0.000,B 0.000,C 90.000,E1 193.119} C_DIS
LIN {X -0.014,Y -482.449,Z 335.864,A 0.000,B 0.000,C 90.000,E1 191.591} C_DIS
LIN {X 0.094,Y -479.155,Z 335.854,A 0.000,B 0.000,C 90.000,E1 189.726} C_DIS
LIN {X 0.128,Y -474.976,Z 335.840,A 0.000,B 0.000,C 90.000,E1 187.239} C_DIS
LIN {X -0.022,Y -471.183,Z 335.826,A 0.000,B 0.000,C 90.000,E1 184.759} C_DIS
LIN {X -0.161,Y -468.266,Z 335.814,A 0.000,B 0.000,C 90.000,E1 182.579} C_DIS
LIN {X 0.047,Y -464.583,Z 335.795,A 0.000,B 0.000,C 90.000,E1 179.083} C_DIS
LIN {X -0.110,Y -461.961,Z 335.774,A 0.000,B 0.000,C 90.000,E1 175.298} C_DIS
LIN {X 0.078,Y -461.062,Z 335.751,A 0.000,B 0.000,C 90.000,E1 171.141} C_DIS
LIN {X -0.062,Y -461.029,Z 335.742,A 0.000,B 0.000,C 90.000,E1 169.567} C_DIS
LIN {X -0.007,Y -461.923,Z 335.723,A 0.000,B 0.000,C 90.000,E1 166.061} C_DIS
LIN {X 0.044,Y -463.506,Z 335.707,A 0.000,B 0.000,C 90.000,E1 163.196} C_DIS
LIN {X 0.172,Y -466.581,Z 335.687,A 0.000,B 0.000,C 90.000,E1 159.699} C_DIS
LIN {X 0.176,Y -471.487,Z 335.666,A 0.000,B 0.000,C 90.000,E1 155.921} C_DIS
LIN {X 0.099,Y -479.375,Z 335.642,A 0.000,B 0.000,C 90.000,E1 151.563} C_DIS
LIN {X 0.051,Y -485.677,Z 335.627,A 0.000,B 0.000,C 90.000,E1 148.791} C_DIS
LIN {X 0.162,Y -493.969,Z 335.610,A 0.000,B 0.000,C 90.000,E1 145.722} C_DIS
LIN {X 0.266,Y -498.346,Z 335.601,A 0.000,B 0.000,C 90.000,E1 144.196} C_DIS
LIN {X 0.157,Y -501.927,Z 335.595,A 0.000,B 0.000,C 90.000,E1 143.004} C_DIS
LIN {X -0.105,Y -506.311,Z 335.586,A 0.000,B 0.000,C 90.000,E1 141.537} C_DIS
LIN {X -0.192,Y -509.522,Z 335.580,A 0.000,B 0.000,C 90.000,E1 140.356} C_DIS
LIN {X -0.147,Y -511.772,Z 335.575,A 0.000,B 0.000,C 90.000,E1 139.461} C_DIS
LIN {X 0.177,Y -514.599,Z 335.568,A 0.000,B 0.000,C 90.000,E1 138.243} C_DIS
LIN {X -0.109,Y -516.291,Z 335.563,A 0.000,B 0.000,C 90.000,E1 137.391} C_DIS
LIN {X -0.021,Y -517.674,Z 335.558,A 0.000,B 0.000,C 90.000,E1 136.500} C_DIS
LIN {X -0.275,Y -518.670,Z 335.553,A 0.000,B 0.000,C 90.000,E1 135.648} C_DIS
LIN {X 0.127,Y -519.520,Z 335.547,A 0.000,B 0.000,C 90.000,E1 134.433} C_DIS
LIN {X 0.252,Y -519.851,Z 335.542,A 0.000,B 0.000,C 90.000,E1 133.542} C_DIS
LIN {X -0.043,Y -519.831,Z 335.536,A 0.000,B 0.000,C 90.000,E1 132.405} C_DIS
LIN {X -0.206,Y -519.547,Z 335.532,A 0.000,B 0.000,C 90.000,E1 131.838} C_DIS
LIN {X 0.013,Y -519.220,Z 335.529,A 0.000,B 0.000,C 90.000,E1 131.229} C_DIS
LIN {X 0.170,Y -518.367,Z 335.524,A 0.000,B 0.000,C 90.000,E1 130.334} C_DIS
LIN {X -0.081,Y -517.353,Z 335.519,A 0.000,B 0.000,C 90.000,E1 129.483} C_DIS
LIN {X -0.153,Y -514.963,Z 335.510,A 0.000,B 0.000,C 90.000,E1 127.729} C_DIS
LIN {X 0.205,Y -512.895,Z 335.501,A 0.000,B 0.000,C 90.000,E1 126.217} C_DIS
LIN {X 0.301,Y -511.064,Z 335.495,A 0.000,B 0.000,C 90.000,E1 125.025} C_DIS
LIN {X -0.247,Y -509.583,Z 335.490,A 0.000,B 0.000,C 90.000,E1 124.199} C_DIS
LIN {X -0.256,Y -506.229,Z 335.480,A 0.000,B 0.000,C 90.000,E1 122.418} C_DIS
LIN {X 0.079,Y -502.484,Z 335.470,A 0.000,B 0.000,C 90.000,E1 120.590} C_DIS
LIN {X 0.206,Y -499.270,Z 335.462,A 0.000,B 0.000,C 90.000,E1 119.077} C_DIS
LIN {X -0.009,Y -496.584,Z 335.455,A 0.000,B 0.000,C 90.000,E1 117.897} C_DIS
LIN {X 0.210,Y -493.187,Z 335.447,A 0.000,B 0.000,C 90.000,E1 116.360} C_DIS
LIN {X 0.154,Y -489.705,Z 335.438,A 0.000,B 0.000,C 90.000,E1 114.847} C_DIS
LIN {X 0.016,Y -486.813,Z 335.431,A 0.000,B 0.000,C 90.000,E1 113.643} C_DIS
LIN {X 0.086,Y -483.775,Z 335.425,A 0.000,B 0.000,C 90.000,E1 112.408} C_DIS
LIN {X 0.112,Y -481.572,Z 335.419,A 0.000,B 0.000,C 90.000,E1 111.482} C_DIS
LIN {X 0.103,Y -478.309,Z 335.413,A 0.000,B 0.000,C 90.000,E1 110.248} C_DIS
LIN {X 0.058,Y -475.838,Z 335.407,A 0.000,B 0.000,C 90.000,E1 109.322} C_DIS
LIN {X 0.054,Y -471.328,Z 335.399,A 0.000,B 0.000,C 90.000,E1 107.764} C_DIS
LIN {X -0.226,Y -468.536,Z 335.394,A 0.000,B 0.000,C 90.000,E1 106.858} C_DIS
LIN {X 0.035,Y -465.443,Z 335.388,A 0.000,B 0.000,C 90.000,E1 105.843} C_DIS
LIN {X -0.006,Y -465.454,Z 335.388,A 0.000,B 0.000,C 90.000,E1 105.843} C_DIS
LIN {X -0.115,Y -467.677,Z 335.383,A 0.000,B 0.000,C 90.000,E1 104.954} C_DIS
LIN {X -0.159,Y -475.891,Z 335.357,A 0.000,B 0.000,C 90.000,E1 100.254} C_DIS
LIN {X 0.149,Y -476.345,Z 335.355,A 0.000,B 0.000,C 90.000,E1 99.905} C_DIS
LIN {X 0.105,Y -481.857,Z 335.331,A 0.000,B 0.000,C 90.000,E1 95.568} C_DIS
LIN {X -0.047,Y -482.188,Z 335.329,A 0.000,B 0.000,C 90.000,E1 95.277} C_DIS
LIN {X -0.113,Y -485.352,Z 335.305,A 0.000,B 0.000,C 90.000,E1 90.974} C_DIS
LIN {X 0.196,Y -485.533,Z 335.304,A 0.000,B 0.000,C 90.000,E1 90.630} C_DIS
LIN {X -0.082,Y -486.340,Z 335.282,A 0.000,B 0.000,C 90.000,E1 86.674} C_DIS
LIN {X 0.053,Y -486.275,Z 335.278,A 0.000,B 0.000,C 90.000,E1 86.045} C_DIS
LIN {X -0.227,Y -484.694,Z 335.254,A 0.000,B 0.000,C 90.000,E1 81.781} C_DIS
LIN {X 0.120,Y -484.548,Z 335.253,A 0.000,B 0.000,C 90.000,E1 81.432} C_DIS
LIN {X -0.010,Y -480.487,Z 335.227,A 0.000,B 0.000,C 90.000,E1 76.825} C_DIS
LIN {X -0.126,Y -477.435,Z 335.216,A 0.000,B 0.000,C 90.000,E1 74.866} C_DIS
LIN {X -0.166,Y -477.447,Z 335.216,A 0.000,B 0.000,C 90.000,E1 74.866} C_DIS
LIN {X 0.042,Y -480.466,Z 335.211,A 0.000,B 0.000,C 90.000,E1 74.031} C_DIS
LIN {X 0.178,Y -484.750,Z 335.204,A 0.000,B 0.000,C 90.000,E1 72.779} C_DIS
LIN {X 0.036,Y -486.803,Z 335.201,A 0.000,B 0.000,C 90.000,E1 72.181} C_DIS
LIN {X -0.076,Y -489.606,Z 335.196,A 0.000,B 0.000,C 90.000,E1 71.275} C_DIS
LIN {X -0.122,Y -493.296,Z 335.189,A 0.000,B 0.000,C 90.000,E1 70.061} C_DIS
LIN {X -0.067,Y -497.794,Z 335.181,A 0.000,B 0.000,C 90.000,E1 68.539} C_DIS
LIN {X -0.282,Y -501.378,Z 335.174,A 0.000,B 0.000,C 90.000,E1 67.358} C_DIS
LIN {X -0.070,Y -506.532,Z 335.164,A 0.000,B 0.000,C 90.000,E1 65.537} C_DIS
LIN {X 0.156,Y -510.793,Z 335.156,A 0.000,B 0.000,C 90.000,E1 64.024} C_DIS
LIN {X -0.116,Y -514.178,Z 335.149,A 0.000,B 0.000,C 90.000,E1 62.871} C_DIS
LIN {X -0.071,Y -519.245,Z 335.139,A 0.000,B 0.000,C 90.000,E1 61.101} C_DIS
LIN {X 0.152,Y -523.408,Z 335.131,A 0.000,B 0.000,C 90.000,E1 59.616} C_DIS
LIN {X -0.199,Y -527.566,Z 335.123,A 0.000,B 0.000,C 90.000,E1 58.201} C_DIS
LIN {X 0.257,Y -531.672,Z 335.115,A 0.000,B 0.000,C 90.000,E1 56.707} C_DIS
LIN {X -0.095,Y -535.610,Z 335.107,A 0.000,B 0.000,C 90.000,E1 55.308} C_DIS
LIN {X 0.047,Y -538.618,Z 335.101,A 0.000,B 0.000,C 90.000,E1 54.149} C_DIS
LIN {X 0.105,Y -541.463,Z 335.095,A 0.000,B 0.000,C 90.000,E1 53.004} C_DIS
LIN {X -0.193,Y -544.668,Z 335.087,A 0.000,B 0.000,C 90.000,E1 51.618} C_DIS
LIN {X -0.089,Y -547.521,Z 335.079,A 0.000,B 0.000,C 90.000,E1 50.194} C_DIS
LIN {X 0.024,Y -549.511,Z 335.073,A 0.000,B 0.000,C 90.000,E1 49.057} C_DIS
LIN {X -0.250,Y -550.848,Z 335.068,A 0.000,B 0.000,C 90.000,E1 48.243} C_DIS
LIN {X 0.277,Y -552.411,Z 335.062,A 0.000,B 0.000,C 90.000,E1 47.067} C_DIS
LIN {X -0.002,Y -553.336,Z 335.057,A 0.000,B 0.000,C 90.000,E1 46.257} C_DIS
LIN {X -0.222,Y -554.231,Z 335.051,A 0.000,B 0.000,C 90.000,E1 45.162} C_DIS
LIN {X 0.303,Y -554.650,Z 335.046,A 0.000,B 0.000,C 90.000,E1 44.271} C_DIS
LIN {X 0.101,Y -554.858,Z 335.040,A 0.000,B 0.000,C 90.000,E1 43.176} C_DIS
LIN {X -0.158,Y -554.798,Z 335.035,A 0.000,B 0.000,C 90.000,E1 42.366} C_DIS
LIN {X 0.051,Y -554.348,Z 335.029,A 0.000,B 0.000,C 90.000,E1 41.229} C_DIS
LIN {X 0.190,Y -553.793,Z 335.024,A 0.000,B 0.000,C 90.000,E1 40.378} C_DIS
LIN {X 0.027,Y -552.789,Z 335.018,A 0.000,B 0.000,C 90.000,E1 39.277} C_DIS
LIN {X -0.144,Y -551.597,Z 335.012,A 0.000,B 0.000,C 90.000,E1 38.177} C_DIS
LIN {X -0.166,Y -549.348,Z 335.001,A 0.000,B 0.000,C 90.000,E1 36.217} C_DIS
LIN {X -0.181,Y -547.288,Z 334.992,A 0.000,B 0.000,C 90.000,E1 34.532} C_DIS
LIN {X -0.027,Y -544.700,Z 334.979,A 0.000,B 0.000,C 90.000,E1 32.260} C_DIS
LIN {X 0.187,Y -542.897,Z 334.970,A 0.000,B 0.000,C 90.000,E1 30.541} C_DIS
LIN {X 0.102,Y -540.736,Z 334.957,A 0.000,B 0.000,C 90.000,E1 28.281} C_DIS
LIN {X -0.014,Y -539.336,Z 334.949,A 0.000,B 0.000,C 90.000,E1 26.873} C_DIS
LIN {X -0.209,Y -537.466,Z 334.938,A 0.000,B 0.000,C 90.000,E1 24.899} C_DIS
LIN {X -0.185,Y -535.694,Z 334.927,A 0.000,B 0.000,C 90.000,E1 22.898} C_DIS
LIN {X 0.088,Y -534.219,Z 334.916,A 0.000,B 0.000,C 90.000,E1 20.865} C_DIS
LIN {X 0.114,Y -533.269,Z 334.906,A 0.000,B 0.000,C 90.000,E1 19.141} C_DIS
LIN {X -0.019,Y -532.124,Z 334.894,A 0.000,B 0.000,C 90.000,E1 16.858} C_DIS
LIN {X 0.144,Y -531.347,Z 334.883,A 0.000,B 0.000,C 90.000,E1 14.828} C_DIS
LIN {X 0.094,Y -530.906,Z 334.868,A 0.000,B 0.000,C 90.000,E1 12.243} C_DIS
LIN {X -0.035,Y -531.197,Z 334.852,A 0.000,B 0.000,C 90.000,E1 9.378} C_DIS
LIN {X 0.101,Y -532.075,Z 334.836,A 0.000,B 0.000,C 90.000,E1 6.486} C_DIS
LIN {X 0.096,Y -532.779,Z 334.828,A 0.000,B 0.000,C 90.000,E1 5.049} C_DIS
LIN {X 0.107,Y -535.020,Z 334.811,A 0.000,B 0.000,C 90.000,E1 1.892} C_DIS
LIN {X 0.219,Y -537.486,Z 334.796,A 0.000,B 0.000,C 90.000,E1 359.198} C_DIS
LIN {X -0.167,Y -540.653,Z 334.781,A 0.000,B 0.000,C 90.000,E1 356.674} C_DIS
LIN {X -0.063,Y -542.176,Z 334.775,A 0.000,B 0.000,C 90.000,E1 355.527} C_DIS
LIN {X 0.103,Y -543.622,Z 334.769,A 0.000,B 0.000,C 90.000,E1 354.375} C_DIS
LIN {X 0.213,Y -544.725,Z 334.764,A 0.000,B 0.000,C 90.000,E1 353.514} C_DIS
LIN {X -0.173,Y -550.210,Z 334.748,A 0.000,B 0.000,C 90.000,E1 350.735} C_DIS
LIN {X -0.251,Y -553.014,Z 334.741,A 0.000,B 0.000,C 90.000,E1 349.342} C_DIS
LIN {X -0.174,Y -556.437,Z 334.733,A 0.000,B 0.000,C 90.000,E1 347.937} C_DIS
LIN {X -0.158,Y -561.896,Z 334.722,A 0.000,B 0.000,C 90.000,E1 345.992} C_DIS
LIN {X -0.174,Y -566.592,Z 334.713,A 0.000,B 0.000,C 90.000,E1 344.338} C_DIS
LIN {X -0.146,Y -572.578,Z 334.702,A 0.000,B 0.000,C 90.000,E1 342.417} C_DIS
LIN {X -0.137,Y -579.420,Z 334.690,A 0.000,B 0.000,C 90.000,E1 340.242} C_DIS
LIN {X 0.187,Y -584.501,Z 334.681,A 0.000,B 0.000,C 90.000,E1 338.592} C_DIS
LIN {X 0.065,Y -589.706,Z 334.672,A 0.000,B 0.000,C 90.000,E1 336.997} C_DIS
LIN {X 0.247,Y -597.848,Z 334.659,A 0.000,B 0.000,C 90.000,E1 334.588} C_DIS
LIN {X -0.132,Y -602.538,Z 334.652,A 0.000,B 0.000,C 90.000,E1 333.307} C_DIS
LIN {X 0.238,Y -609.941,Z 334.640,A 0.000,B 0.000,C 90.000,E1 331.179} C_DIS
LIN {X 0.009,Y -618.541,Z 334.627,A 0.000,B 0.000,C 90.000,E1 328.869} C_DIS
LIN {X 0.041,Y -623.115,Z 334.620,A 0.000,B 0.000,C 90.000,E1 327.582} C_DIS
LIN {X 0.156,Y -626.646,Z 334.614,A 0.000,B 0.000,C 90.000,E1 326.548} C_DIS
LIN {X -0.032,Y -629.056,Z 334.610,A 0.000,B 0.000,C 90.000,E1 325.801} C_DIS
LIN {X 0.010,Y -632.851,Z 334.603,A 0.000,B 0.000,C 90.000,E1 324.529} C_DIS
LIN {X 0.117,Y -636.533,Z 334.596,A 0.000,B 0.000,C 90.000,E1 323.256} C_DIS
LIN {X 0.072,Y -642.058,Z 334.585,A 0.000,B 0.000,C 90.000,E1 321.251} C_DIS
LIN {X 0.057,Y -647.915,Z 334.574,A 0.000,B 0.000,C 90.000,E1 319.256} C_DIS
LIN {X -0.314,Y -653.007,Z 334.564,A 0.000,B 0.000,C 90.000,E1 317.553} C_DIS
LIN {X -0.144,Y -659.253,Z 334.553,A 0.000,B 0.000,C 90.000,E1 315.567} C_DIS
LIN {X -0.230,Y -662.320,Z 334.548,A 0.000,B 0.000,C 90.000,E1 314.595} C_DIS
LIN {X 0.193,Y -666.769,Z 334.540,A 0.000,B 0.000,C 90.000,E1 313.095} C_DIS
LIN {X -0.251,Y -670.314,Z 334.533,A 0.000,B 0.000,C 90.000,E1 311.919} C_DIS
LIN {X 0.286,Y -672.958,Z 334.527,A 0.000,B 0.000,C 90.000,E1 310.906} C_DIS
LIN {X -0.019,Y -675.434,Z 334.522,A 0.000,B 0.000,C 90.000,E1 309.967} C_DIS
LIN {X -0.396,Y -677.261,Z 334.518,A 0.000,B 0.000,C 90.000,E1 309.277} C_DIS
LIN {X -0.216,Y -679.518,Z 334.513,A 0.000,B 0.000,C 90.000,E1 308.302} C_DIS
LIN {X 0.110,Y -681.493,Z 334.507,A 0.000,B 0.000,C 90.000,E1 307.317} C_DIS
LIN {X 0.310,Y -682.854,Z 334.503,A 0.000,B 0.000,C 90.000,E1 306.583} C_DIS
LIN {X 0.116,Y -683.995,Z 334.499,A 0.000,B 0.000,C 90.000,E1 305.884} C_DIS
LIN {X -0.246,Y -684.760,Z 334.497,A 0.000,B 0.000,C 90.000,E1 305.438} C_DIS
LIN {X -0.237,Y -685.824,Z 334.492,A 0.000,B 0.000,C 90.000,E1 304.485} C_DIS
LIN {X -0.030,Y -686.269,Z 334.489,A 0.000,B 0.000,C 90.000,E1 303.992} C_DIS
LIN {X -0.195,Y -686.699,Z 334.485,A 0.000,B 0.000,C 90.000,E1 303.293} C_DIS
LIN {X 0.011,Y -686.846,Z 334.482,A 0.000,B 0.000,C 90.000,E1 302.801} C_DIS
LIN {X 0.057,Y -686.772,Z 334.478,A 0.000,B 0.000,C 90.000,E1 302.084} C_DIS
LIN {X 0.098,Y -686.247,Z 334.473,A 0.000,B 0.000,C 90.000,E1 301.131} C_DIS
LIN {X 0.153,Y -685.590,Z 334.469,A 0.000,B 0.000,C 90.000,E1 300.413} C_DIS
LIN {X -0.047,Y -684.680,Z 334.465,A 0.000,B 0.000,C 90.000,E1 299.716} C_DIS
LIN {X -0.007,Y -683.505,Z 334.461,A 0.000,B 0.000,C 90.000,E1 298.999} C_DIS
LIN {X 0.229,Y -681.653,Z 334.456,A 0.000,B 0.000,C 90.000,E1 298.025} C_DIS
LIN {X 0.131,Y -679.549,Z 334.451,A 0.000,B 0.000,C 90.000,E1 297.078} C_DIS
LIN {X 0.318,Y -677.331,Z 334.445,A 0.000,B 0.000,C 90.000,E1 296.104} C_DIS
LIN {X -0.253,Y -674.333,Z 334.439,A 0.000,B 0.000,C 90.000,E1 294.951} C_DIS
LIN {X 0.244,Y -670.507,Z 334.431,A 0.000,B 0.000,C 90.000,E1 293.462} C_DIS
LIN {X -0.094,Y -667.092,Z 334.424,A 0.000,B 0.000,C 90.000,E1 292.280} C_DIS
LIN {X 0.279,Y -661.761,Z 334.413,A 0.000,B 0.000,C 90.000,E1 290.301} C_DIS
LIN {X 0.051,Y -656.745,Z 334.402,A 0.000,B 0.000,C 90.000,E1 288.362} C_DIS
LIN {X 0.123,Y -652.036,Z 334.391,A 0.000,B 0.000,C 90.000,E1 286.386} C_DIS
LIN {X 0.061,Y -647.765,Z 334.380,A 0.000,B 0.000,C 90.000,E1 284.411} C_DIS
LIN {X 0.222,Y -642.719,Z 334.365,A 0.000,B 0.000,C 90.000,E1 281.658} C_DIS
LIN {X 0.098,Y -638.882,Z 334.350,A 0.000,B 0.000,C 90.000,E1 278.916} C_DIS
LIN {X 0.146,Y -635.660,Z 334.330,A 0.000,B 0.000,C 90.000,E1 275.391} C_DIS
LIN {X 0.056,Y -634.188,Z 334.312,A 0.000,B 0.000,C 90.000,E1 272.121} C_DIS
LIN {X -0.115,Y -633.963,Z 334.294,A 0.000,B 0.000,C 90.000,E1 268.854} C_DIS
LIN {X -0.123,Y -634.806,Z 334.280,A 0.000,B 0.000,C 90.000,E1 266.331} C_DIS
LIN {X -0.170,Y -635.895,Z 334.268,A 0.000,B 0.000,C 90.000,E1 264.318} C_DIS
LIN {X -0.122,Y -637.329,Z 334.257,A 0.000,B 0.000,C 90.000,E1 262.299} C_DIS
LIN {X 0.041,Y -638.986,Z 334.246,A 0.000,B 0.000,C 90.000,E1 260.274} C_DIS
LIN {X 0.004,Y -640.747,Z 334.236,A 0.000,B 0.000,C 90.000,E1 258.522} C_DIS
LIN {X 0.001,Y -643.216,Z 334.225,A 0.000,B 0.000,C 90.000,E1 256.520} C_DIS
LIN {X 0.025,Y -644.452,Z 334.220,A 0.000,B 0.000,C 90.000,E1 255.519} C_DIS
LIN {X 0.205,Y -645.151,Z 334.215,A 0.000,B 0.000,C 90.000,E1 254.755} C_DIS
LIN {X 0.268,Y -646.040,Z 334.209,A 0.000,B 0.000,C 90.000,E1 253.504} C_DIS
LIN {X -0.276,Y -646.479,Z 334.202,A 0.000,B 0.000,C 90.000,E1 252.308} C_DIS
LIN {X 0.241,Y -646.632,Z 334.199,A 0.000,B 0.000,C 90.000,E1 251.764} C_DIS
LIN {X 0.057,Y -646.374,Z 334.193,A 0.000,B 0.000,C 90.000,E1 250.786} C_DIS
LIN {X -0.096,Y -646.300,Z 334.192,A 0.000,B 0.000,C 90.000,E1 250.550} C_DIS
LIN {X -0.123,Y -645.660,Z 334.188,A 0.000,B 0.000,C 90.000,E1 249.806} C_DIS
LIN {X 0.390,Y -645.113,Z 334.185,A 0.000,B 0.000,C 90.000,E1 249.263} C_DIS
LIN {X 0.123,Y -643.923,Z 334.181,A 0.000,B 0.000,C 90.000,E1 248.539} C_DIS
LIN {X 0.014,Y -643.023,Z 334.178,A 0.000,B 0.000,C 90.000,E1 248.050} C_DIS
LIN {X 0.021,Y -640.791,Z 334.173,A 0.000,B 0.000,C 90.000,E1 247.050} C_DIS
LIN {X 0.143,Y -639.541,Z 334.170,A 0.000,B 0.000,C 90.000,E1 246.538} C_DIS
LIN {X 0.058,Y -637.498,Z 334.166,A 0.000,B 0.000,C 90.000,E1 245.793} C_DIS
LIN {X -0.053,Y -635.424,Z 334.161,A 0.000,B 0.000,C 90.000,E1 245.049} C_DIS
LIN {X 0.122,Y -632.189,Z 334.156,A 0.000,B 0.000,C 90.000,E1 244.024} C_DIS
LIN {X 0.283,Y -627.853,Z 334.149,A 0.000,B 0.000,C 90.000,E1 242.743} C_DIS
LIN {X -0.180,Y -622.471,Z 334.140,A 0.000,B 0.000,C 90.000,E1 241.257} C_DIS
LIN {X 0.101,Y -618.057,Z 334.133,A 0.000,B 0.000,C 90.000,E1 239.950} C_DIS
LIN {X 0.333,Y -611.764,Z 334.123,A 0.000,B 0.000,C 90.000,E1 238.122} C_DIS
LIN {X 0.220,Y -607.254,Z 334.116,A 0.000,B 0.000,C 90.000,E1 236.834} C_DIS
LIN {X 0.022,Y -602.601,Z 334.109,A 0.000,B 0.000,C 90.000,E1 235.548} C_DIS
LIN {X 0.295,Y -595.269,Z 334.097,A 0.000,B 0.000,C 90.000,E1 233.417} C_DIS
LIN {X 0.138,Y -592.431,Z 334.093,A 0.000,B 0.000,C 90.000,E1 232.637} C_DIS
LIN {X 0.017,Y -584.716,Z 334.081,A 0.000,B 0.000,C 90.000,E1 230.517} C_DIS
LIN {X 0.009,Y -580.102,Z 334.073,A 0.000,B 0.000,C 90.000,E1 229.175} C_DIS
LIN {X -0.276,Y -573.805,Z 334.063,A 0.000,B 0.000,C 90.000,E1 227.310} C_DIS
LIN {X -0.216,Y -570.202,Z 334.057,A 0.000,B 0.000,C 90.000,E1 226.215} C_DIS
LIN {X 0.054,Y -563.885,Z 334.046,A 0.000,B 0.000,C 90.000,E1 224.271} C_DIS
LIN {X -0.153,Y -556.730,Z 334.034,A 0.000,B 0.000,C 90.000,E1 222.081} C_DIS
LIN {X -0.156,Y -549.597,Z 334.021,A 0.000,B 0.000,C 90.000,E1 219.850} C_DIS
LIN {X 0.047,Y -546.172,Z 334.015,A 0.000,B 0.000,C 90.000,E1 218.705} C_DIS
LIN {X -0.126,Y -540.149,Z 334.004,A 0.000,B 0.000,C 90.000,E1 216.744} C_DIS
LIN {X -0.031,Y -535.346,Z 333.995,A 0.000,B 0.000,C 90.000,E1 215.025} C_DIS
LIN {X -0.246,Y -529.122,Z 333.982,A 0.000,B 0.000,C 90.000,E1 212.752} C_DIS
LIN {X -0.020,Y -523.552,Z 333.969,A 0.000,B 0.000,C 90.000,E1 210.413} C_DIS
LIN {X -0.266,Y -519.486,Z 333.959,A 0.000,B 0.000,C 90.000,E1 208.693} C_DIS
LIN {X -0.157,Y -515.522,Z 333.950,A 0.000,B 0.000,C 90.000,E1 206.924} C_DIS
LIN {X -0.145,Y -511.638,Z 333.940,A 0.000,B 0.000,C 90.000,E1 205.155} C_DIS
LIN {X 0.044,Y -509.050,Z 333.933,A 0.000,B 0.000,C 90.000,E1 203.951} C_DIS
LIN {X 0.084,Y -505.729,Z 333.925,A 0.000,B 0.000,C 90.000,E1 202.461} C_DIS
LIN {X 0.059,Y -502.378,Z 333.917,A 0.000,B 0.000,C 90.000,E1 200.972} C_DIS
LIN {X 0.190,Y -499.717,Z 333.910,A 0.000,B 0.000,C 90.000,E1 199.758} C_DIS
LIN {X -0.236,Y -495.746,Z 333.900,A 0.000,B 0.000,C 90.000,E1 198.000} C_DIS
LIN {X -0.012,Y -490.210,Z 333.885,A 0.000,B 0.000,C 90.000,E1 195.245} C_DIS
LIN {X -0.110,Y -486.187,Z 333.873,A 0.000,B 0.000,C 90.000,E1 193.119} C_DIS
LIN {X -0.159,Y -483.409,Z 333.864,A 0.000,B 0.000,C 90.000,E1 191.591} C_DIS
LIN {X 0.113,Y -480.694,Z 333.856,A 0.000,B 0.000,C 90.000,E1 190.018} C_DIS
LIN {X -0.053,Y -477.016,Z 333.844,A 0.000,B 0.000,C 90.000,E1 187.871} C_DIS
LIN {X 0.033,Y -473.595,Z 333.832,A 0.000,B 0.000,C 90.000,E1 185.682} C_DIS
LIN {X -0.231,Y -470.170,Z 333.818,A 0.000,B 0.000,C 90.000,E1 183.212} C_DIS
LIN {X 0.064,Y -465.669,Z 333.795,A 0.000,B 0.000,C 90.000,E1 179.083} C_DIS
LIN {X 0.211,Y -463.206,Z 333.776,A 0.000,B 0.000,C 90.000,E1 175.584} C_DIS
LIN {X 0.159,Y -462.137,Z 333.754,A 0.000,B 0.000,C 90.000,E1 171.781} C_DIS
LIN {X -0.172,Y -462.120,Z 333.744,A 0.000,B 0.000,C 90.000,E1 169.916} C_DIS
LIN {X 0.083,Y -463.105,Z 333.721,A 0.000,B 0.000,C 90.000,E1 165.755} C_DIS
LIN {X -0.103,Y -464.313,Z 333.709,A 0.000,B 0.000,C 90.000,E1 163.559} C_DIS
LIN {X 0.115,Y -466.859,Z 333.691,A 0.000,B 0.000,C 90.000,E1 160.369} C_DIS
LIN {X 0.127,Y -469.737,Z 333.677,A 0.000,B 0.000,C 90.000,E1 157.847} C_DIS
LIN {X 0.032,Y -475.356,Z 333.656,A 0.000,B 0.000,C 90.000,E1 154.101} C_DIS
LIN {X -0.016,Y -481.462,Z 333.639,A 0.000,B 0.000,C 90.000,E1 151.001} C_DIS
LIN {X -0.229,Y -486.366,Z 333.627,A 0.000,B 0.000,C 90.000,E1 148.869} C_DIS
LIN {X -0.050,Y -491.930,Z 333.615,A 0.000,B 0.000,C 90.000,E1 146.707} C_DIS
LIN {X -0.131,Y -497.076,Z 333.605,A 0.000,B 0.000,C 90.000,E1 144.895} C_DIS
LIN {X 0.198,Y -502.266,Z 333.595,A 0.000,B 0.000,C 90.000,E1 143.050} C_DIS
LIN {X -0.052,Y -506.540,Z 333.587,A 0.000,B 0.000,C 90.000,E1 141.582} C_DIS
LIN {X 0.264,Y -509.581,Z 333.580,A 0.000,B 0.000,C 90.000,E1 140.356} C_DIS
LIN {X 0.312,Y -511.795,Z 333.575,A 0.000,B 0.000,C 90.000,E1 139.461} C_DIS
LIN {X -0.088,Y -514.476,Z 333.568,A 0.000,B 0.000,C 90.000,E1 138.324} C_DIS
LIN {X -0.027,Y -516.152,Z 333.564,A 0.000,B 0.000,C 90.000,E1 137.433} C_DIS
LIN {X 0.083,Y -517.530,Z 333.559,A 0.000,B 0.000,C 90.000,E1 136.539} C_DIS
LIN {X 0.185,Y -518.468,Z 333.554,A 0.000,B 0.000,C 90.000,E1 135.648} C_DIS
LIN {X -0.068,Y -519.096,Z 333.549,A 0.000,B 0.000,C 90.000,E1 134.798} C_DIS
LIN {X -0.313,Y -519.485,Z 333.544,A 0.000,B 0.000,C 90.000,E1 133.947} C_DIS
LIN {X 0.188,Y -519.538,Z 333.539,A 0.000,B 0.000,C 90.000,E1 133.014} C_DIS
LIN {X -0.042,Y -519.288,Z 333.534,A 0.000,B 0.000,C 90.000,E1 132.162} C_DIS
LIN {X 0.067,Y -518.704,Z 333.529,A 0.000,B 0.000,C 90.000,E1 131.272} C_DIS
LIN {X 0.147,Y -517.456,Z 333.523,A 0.000,B 0.000,C 90.000,E1 130.092} C_DIS
LIN {X 0.283,Y -516.356,Z 333.518,A 0.000,B 0.000,C 90.000,E1 129.197} C_DIS
LIN {X 0.191,Y -513.974,Z 333.508,A 0.000,B 0.000,C 90.000,E1 127.443} C_DIS
LIN {X -0.108,Y -512.285,Z 333.502,A 0.000,B 0.000,C 90.000,E1 126.297} C_DIS
LIN {X -0.017,Y -510.474,Z 333.495,A 0.000,B 0.000,C 90.000,E1 125.105} C_DIS
LIN {X 0.045,Y -508.389,Z 333.488,A 0.000,B 0.000,C 90.000,E1 123.913} C_DIS
LIN {X 0.112,Y -505.592,Z 333.480,A 0.000,B 0.000,C 90.000,E1 122.418} C_DIS
LIN {X 0.126,Y -502.511,Z 333.472,A 0.000,B 0.000,C 90.000,E1 120.924} C_DIS
LIN {X -0.041,Y -500.010,Z 333.465,A 0.000,B 0.000,C 90.000,E1 119.745} C_DIS
LIN {X 0.043,Y -496.704,Z 333.457,A 0.000,B 0.000,C 90.000,E1 118.231} C_DIS
LIN {X 0.085,Y -492.701,Z 333.447,A 0.000,B 0.000,C 90.000,E1 116.411} C_DIS
LIN {X 0.043,Y -488.600,Z 333.437,A 0.000,B 0.000,C 90.000,E1 114.591} C_DIS
LIN {X -0.097,Y -485.032,Z 333.428,A 0.000,B 0.000,C 90.000,E1 113.078} C_DIS
LIN {X -0.049,Y -480.636,Z 333.418,A 0.000,B 0.000,C 90.000,E1 111.227} C_DIS
LIN {X -0.064,Y -478.224,Z 333.413,A 0.000,B 0.000,C 90.000,E1 110.301} C_DIS
LIN {X 0.158,Y -474.964,Z 333.406,A 0.000,B 0.000,C 90.000,E1 109.033} C_DIS
LIN {X -0.160,Y -470.601,Z 333.397,A 0.000,B 0.000,C 90.000,E1 107.511} C_DIS
LIN {X -0.005,Y -467.874,Z 333.392,A 0.000,B 0.000,C 90.000,E1 106.551} C_DIS
LIN {X 0.000,Y -465.593,Z 333.388,A 0.000,B 0.000,C 90.000,E1 105.788} C_DIS
LIN {X -0.040,Y -465.596,Z 333.388,A 0.000,B 0.000,C 90.000,E1 105.788} C_DIS
LIN {X 0.165,Y -467.590,Z 333.383,A 0.000,B 0.000,C 90.000,E1 104.954} C_DIS
LIN {X -0.103,Y -468.589,Z 333.380,A 0.000,B 0.000,C 90.000,E1 104.356} C_DIS
LIN {X 0.124,Y -475.819,Z 333.357,A 0.000,B 0.000,C 90.000,E1 100.254} C_DIS
LIN {X -0.038,Y -476.313,Z 333.355,A 0.000,B 0.000,C 90.000,E1 99.962} C_DIS
LIN {X -0.091,Y -481.802,Z 333.331,A 0.000,B 0.000,C 90.000,E1 95.625} C_DIS
LIN {X 0.236,Y -482.175,Z 333.330,A 0.000,B 0.000,C 90.000,E1 95.277} C_DIS
LIN {X 0.170,Y -485.317,Z 333.306,A 0.000,B 0.000,C 90.000,E1 90.974} C_DIS
LIN {X -0.005,Y -485.536,Z 333.304,A 0.000,B 0.000,C 90.000,E1 90.688} C_DIS
LIN {X 0.202,Y -486.323,Z 333.282,A 0.000,B 0.000,C 90.000,E1 86.674} C_DIS
LIN {X -0.148,Y -486.299,Z 333.278,A 0.000,B 0.000,C 90.000,E1 86.102} C_DIS
LIN {X 0.056,Y -484.696,Z 333.254,A 0.000,B 0.000,C 90.000,E1 81.781} C_DIS
LIN {X -0.075,Y -484.590,Z 333.253,A 0.000,B 0.000,C 90.000,E1 81.489} C_DIS
LIN {X -0.195,Y -480.526,Z 333.227,A 0.000,B 0.000,C 90.000,E1 76.881} C_DIS
LIN {X 0.091,Y -477.395,Z 333.216,A 0.000,B 0.000,C 90.000,E1 74.810} C_DIS
LIN {X 0.051,Y -477.412,Z 333.216,A 0.000,B 0.000,C 90.000,E1 74.810} C_DIS
LIN {X -0.271,Y -480.176,Z 333.212,A 0.000,B 0.000,C 90.000,E1 74.102} C_DIS
LIN {X 0.000,Y -483.352,Z 333.206,A 0.000,B 0.000,C 90.000,E1 73.142} C_DIS
LIN {X -0.151,Y -486.333,Z 333.201,A 0.000,B 0.000,C 90.000,E1 72.236} C_DIS
LIN {X 0.197,Y -489.057,Z 333.196,A 0.000,B 0.000,C 90.000,E1 71.275} C_DIS
LIN {X 0.143,Y -492.623,Z 333.189,A 0.000,B 0.000,C 90.000,E1 70.061} C_DIS
LIN {X 0.188,Y -497.055,Z 333.181,A 0.000,B 0.000,C 90.000,E1 68.539} C_DIS
LIN {X -0.036,Y -500.616,Z 333.174,A 0.000,B 0.000,C 90.000,E1 67.358} C_DIS
LIN {X 0.246,Y -506.596,Z 333.163,A 0.000,B 0.000,C 90.000,E1 65.229} C_DIS
LIN {X 0.013,Y -510.847,Z 333.154,A 0.000,B 0.000,C 90.000,E1 63.768} C_DIS
LIN {X -0.259,Y -514.252,Z 333.148,A 0.000,B 0.000,C 90.000,E1 62.615} C_DIS
LIN {X 0.239,Y -519.332,Z 333.138,A 0.000,B 0.000,C 90.000,E1 60.795} C_DIS
LIN {X -0.111,Y -525.198,Z 333.127,A 0.000,B 0.000,C 90.000,E1 58.791} C_DIS
LIN {X -0.007,Y -530.161,Z 333.117,A 0.000,B 0.000,C 90.000,E1 57.041} C_DIS
LIN {X 0.048,Y -534.954,Z 333.107,A 0.000,B 0.000,C 90.000,E1 55.308} C_DIS
LIN {X -0.254,Y -537.951,Z 333.101,A 0.000,B 0.000,C 90.000,E1 54.196} C_DIS
LIN {X -0.181,Y -541.511,Z 333.093,A 0.000,B 0.000,C 90.000,E1 52.763} C_DIS
LIN {X -0.048,Y -544.678,Z 333.085,A 0.000,B 0.000,C 90.000,E1 51.331} C_DIS
LIN {X 0.056,Y -547.494,Z 333.077,A 0.000,B 0.000,C 90.000,E1 49.908} C_DIS
LIN {X 0.209,Y -549.921,Z 333.070,A 0.000,B 0.000,C 90.000,E1 48.485} C_DIS
LIN {X -0.014,Y -551.945,Z 333.062,A 0.000,B 0.000,C 90.000,E1 47.106} C_DIS
LIN {X 0.124,Y -553.234,Z 333.056,A 0.000,B 0.000,C 90.000,E1 45.972} C_DIS
LIN {X -0.147,Y -553.944,Z 333.051,A 0.000,B 0.000,C 90.000,E1 45.162} C_DIS
LIN {X -0.022,Y -554.418,Z 333.046,A 0.000,B 0.000,C 90.000,E1 44.312} C_DIS
LIN {X 0.170,Y -554.676,Z 333.040,A 0.000,B 0.000,C 90.000,E1 43.176} C_DIS
LIN {X -0.092,Y -554.661,Z 333.035,A 0.000,B 0.000,C 90.000,E1 42.366} C_DIS
LIN {X 0.051,Y -554.393,Z 333.031,A 0.000,B 0.000,C 90.000,E1 41.515} C_DIS
LIN {X -0.173,Y -553.998,Z 333.026,A 0.000,B 0.000,C 90.000,E1 40.701} C_DIS
LIN {X 0.025,Y -553.147,Z 333.020,A 0.000,B 0.000,C 90.000,E1 39.564} C_DIS
LIN {X -0.143,Y -552.094,Z 333.014,A 0.000,B 0.000,C 90.000,E1 38.463} C_DIS
LIN {X -0.210,Y -550.207,Z 333.004,A 0.000,B 0.000,C 90.000,E1 36.790} C_DIS
LIN {X -0.042,Y -549.303,Z 333.000,A 0.000,B 0.000,C 90.000,E1 35.931} C_DIS
LIN {X -0.060,Y -547.265,Z 332.990,A 0.000,B 0.000,C 90.000,E1 34.246} C_DIS
LIN {X 0.057,Y -545.049,Z 332.979,A 0.000,B 0.000,C 90.000,E1 32.260} C_DIS
LIN {X -0.189,Y -543.307,Z 332.970,A 0.000,B 0.000,C 90.000,E1 30.590} C_DIS
LIN {X -0.050,Y -541.156,Z 332.957,A 0.000,B 0.000,C 90.000,E1 28.309} C_DIS
LIN {X -0.168,Y -539.511,Z 332.948,A 0.000,B 0.000,C 90.000,E1 26.616} C_DIS
LIN {X -0.087,Y -537.954,Z 332.938,A 0.000,B 0.000,C 90.000,E1 24.899} C_DIS
LIN {X -0.121,Y -535.708,Z 332.924,A 0.000,B 0.000,C 90.000,E1 22.333} C_DIS
LIN {X -0.131,Y -534.085,Z 332.910,A 0.000,B 0.000,C 90.000,E1 19.758} C_DIS
LIN {X -0.263,Y -532.992,Z 332.899,A 0.000,B 0.000,C 90.000,E1 17.764} C_DIS
LIN {X 0.113,Y -532.089,Z 332.886,A 0.000,B 0.000,C 90.000,E1 15.426} C_DIS
LIN {X -0.266,Y -531.408,Z 332.870,A 0.000,B 0.000,C 90.000,E1 12.591} C_DIS
LIN {X 0.142,Y -531.587,Z 332.854,A 0.000,B 0.000,C 90.000,E1 9.670} C_DIS
LIN {X -0.234,Y -532.128,Z 332.841,A 0.000,B 0.000,C 90.000,E1 7.409} C_DIS
LIN {X -0.208,Y -532.888,Z 332.831,A 0.000,B 0.000,C 90.000,E1 5.682} C_DIS
LIN {X -0.167,Y -534.614,Z 332.816,A 0.000,B 0.000,C 90.000,E1 2.808} C_DIS
LIN {X -0.154,Y -536.005,Z 332.806,A 0.000,B 0.000,C 90.000,E1 1.088} C_DIS
LIN {X 0.230,Y -537.917,Z 332.794,A 0.000,B 0.000,C 90.000,E1 358.912} C_DIS
LIN {X -0.145,Y -541.024,Z 332.780,A 0.000,B 0.000,C 90.000,E1 356.388} C_DIS
LIN {X -0.058,Y -542.112,Z 332.775,A 0.000,B 0.000,C 90.000,E1 355.527} C_DIS
LIN {X 0.125,Y -543.849,Z 332.767,A 0.000,B 0.000,C 90.000,E1 354.090} C_DIS
LIN {X -0.246,Y -545.028,Z 332.763,A 0.000,B 0.000,C 90.000,E1 353.280} C_DIS
LIN {X -0.176,Y -550.004,Z 332.748,A 0.000,B 0.000,C 90.000,E1 350.735} C_DIS
LIN {X 0.105,Y -554.735,Z 332.736,A 0.000,B 0.000,C 90.000,E1 348.465} C_DIS
LIN {X -0.175,Y -561.644,Z 332.722,A 0.000,B 0.000,C 90.000,E1 345.992} C_DIS
LIN {X -0.197,Y -566.341,Z 332.713,A 0.000,B 0.000,C 90.000,E1 344.338} C_DIS
LIN {X -0.174,Y -572.304,Z 332.702,A 0.000,B 0.000,C 90.000,E1 342.417} C_DIS
LIN {X -0.175,Y -579.141,Z 332.690,A 0.000,B 0.000,C 90.000,E1 340.242} C_DIS
LIN {X 0.144,Y -584.223,Z 332.681,A 0.000,B 0.000,C 90.000,E1 338.592} C_DIS
LIN {X 0.246,Y -589.426,Z 332.672,A 0.000,B 0.000,C 90.000,E1 336.975} C_DIS
LIN {X 0.187,Y -597.568,Z 332.659,A 0.000,B 0.000,C 90.000,E1 334.588} C_DIS
LIN {X 0.342,Y -602.259,Z 332.652,A 0.000,B 0.000,C 90.000,E1 333.256} C_DIS
LIN {X 0.165,Y -609.661,Z 332.640,A 0.000,B 0.000,C 90.000,E1 331.179} C_DIS
LIN {X -0.074,Y -618.265,Z 332.627,A 0.000,B 0.000,C 90.000,E1 328.869} C_DIS
LIN {X -0.047,Y -622.841,Z 332.620,A 0.000,B 0.000,C 90.000,E1 327.582} C_DIS
LIN {X 0.064,Y -626.368,Z 332.614,A 0.000,B 0.000,C 90.000,E1 326.548} C_DIS
LIN {X -0.126,Y -628.776,Z 332.610,A 0.000,B 0.000,C 90.000,E1 325.801} C_DIS
LIN {X -0.091,Y -632.574,Z 332.603,A 0.000,B 0.000,C 90.000,E1 324.529} C_DIS
LIN {X 0.012,Y -636.253,Z 332.596,A 0.000,B 0.000,C 90.000,E1 323.256} C_DIS
LIN {X 0.059,Y -641.057,Z 332.586,A 0.000,B 0.000,C 90.000,E1 321.492} C_DIS
LIN {X -0.232,Y -643.906,Z 332.581,A 0.000,B 0.000,C 90.000,E1 320.517} C_DIS
LIN {X -0.137,Y -648.345,Z 332.572,A 0.000,B 0.000,C 90.000,E1 319.013} C_DIS
LIN {X -0.015,Y -653.442,Z 332.563,A 0.000,B 0.000,C 90.000,E1 317.268} C_DIS
LIN {X -0.284,Y -658.920,Z 332.553,A 0.000,B 0.000,C 90.000,E1 315.567} C_DIS
LIN {X -0.376,Y -661.976,Z 332.548,A 0.000,B 0.000,C 90.000,E1 314.595} C_DIS
LIN {X 0.044,Y -665.680,Z 332.541,A 0.000,B 0.000,C 90.000,E1 313.338} C_DIS
LIN {X 0.036,Y -669.218,Z 332.534,A 0.000,B 0.000,C 90.000,E1 312.123} C_DIS
LIN {X 0.111,Y -671.898,Z 332.529,A 0.000,B 0.000,C 90.000,E1 311.148} C_DIS
LIN {X -0.298,Y -673.763,Z 332.525,A 0.000,B 0.000,C 90.000,E1 310.458} C_DIS
LIN {X 0.379,Y -676.788,Z 332.518,A 0.000,B 0.000,C 90.000,E1 309.197} C_DIS
LIN {X 0.004,Y -678.456,Z 332.514,A 0.000,B 0.000,C 90.000,E1 308.508} C_DIS
LIN {X 0.312,Y -680.477,Z 332.509,A 0.000,B 0.000,C 90.000,E1 307.523} C_DIS
LIN {X 0.114,Y -682.246,Z 332.503,A 0.000,B 0.000,C 90.000,E1 306.583} C_DIS
LIN {X -0.071,Y -683.699,Z 332.498,A 0.000,B 0.000,C 90.000,E1 305.644} C_DIS
LIN {X 0.301,Y -684.598,Z 332.494,A 0.000,B 0.000,C 90.000,E1 304.898} C_DIS
LIN {X 0.124,Y -685.327,Z 332.490,A 0.000,B 0.000,C 90.000,E1 304.199} C_DIS
LIN {X 0.150,Y -685.854,Z 332.485,A 0.000,B 0.000,C 90.000,E1 303.245} C_DIS
LIN {X 0.353,Y -685.988,Z 332.482,A 0.000,B 0.000,C 90.000,E1 302.752} C_DIS
LIN {X -0.186,Y -685.861,Z 332.478,A 0.000,B 0.000,C 90.000,E1 302.084} C_DIS
LIN {X 0.220,Y -685.458,Z 332.474,A 0.000,B 0.000,C 90.000,E1 301.337} C_DIS
LIN {X -0.322,Y -684.846,Z 332.470,A 0.000,B 0.000,C 90.000,E1 300.669} C_DIS
LIN {X 0.065,Y -683.961,Z 332.466,A 0.000,B 0.000,C 90.000,E1 299.922} C_DIS
LIN {X 0.099,Y -682.860,Z 332.462,A 0.000,B 0.000,C 90.000,E1 299.205} C_DIS
LIN {X 0.125,Y -681.526,Z 332.458,A 0.000,B 0.000,C 90.000,E1 298.487} C_DIS
LIN {X 0.338,Y -679.489,Z 332.453,A 0.000,B 0.000,C 90.000,E1 297.513} C_DIS
LIN {X -0.195,Y -676.704,Z 332.446,A 0.000,B 0.000,C 90.000,E1 296.360} C_DIS
LIN {X -0.162,Y -673.715,Z 332.440,A 0.000,B 0.000,C 90.000,E1 295.155} C_DIS
LIN {X -0.179,Y -670.543,Z 332.433,A 0.000,B 0.000,C 90.000,E1 293.951} C_DIS
LIN {X 0.200,Y -667.880,Z 332.428,A 0.000,B 0.000,C 90.000,E1 292.950} C_DIS
LIN {X -0.161,Y -663.062,Z 332.418,A 0.000,B 0.000,C 90.000,E1 291.280} C_DIS
LIN {X -0.130,Y -659.149,Z 332.410,A 0.000,B 0.000,C 90.000,E1 289.812} C_DIS
LIN {X 0.316,Y -654.836,Z 332.401,A 0.000,B 0.000,C 90.000,E1 288.055} C_DIS
LIN {X 0.198,Y -649.671,Z 332.388,A 0.000,B 0.000,C 90.000,E1 285.843} C_DIS
LIN {X -0.098,Y -645.476,Z 332.377,A 0.000,B 0.000,C 90.000,E1 283.883} C_DIS
LIN {X -0.011,Y -640.696,Z 332.362,A 0.000,B 0.000,C 90.000,E1 281.130} C_DIS
LIN {X -0.313,Y -637.064,Z 332.347,A 0.000,B 0.000,C 90.000,E1 278.398} C_DIS
LIN {X 0.137,Y -634.463,Z 332.330,A 0.000,B 0.000,C 90.000,E1 275.334} C_DIS
LIN {X -0.001,Y -633.007,Z 332.312,A 0.000,B 0.000,C 90.000,E1 272.064} C_DIS
LIN {X -0.069,Y -632.716,Z 332.297,A 0.000,B 0.000,C 90.000,E1 269.542} C_DIS
LIN {X 0.013,Y -633.068,Z 332.288,A 0.000,B 0.000,C 90.000,E1 267.764} C_DIS
LIN {X 0.244,Y -634.058,Z 332.275,A 0.000,B 0.000,C 90.000,E1 265.469} C_DIS
LIN {X 0.170,Y -635.326,Z 332.264,A 0.000,B 0.000,C 90.000,E1 263.457} C_DIS
LIN {X 0.110,Y -636.458,Z 332.255,A 0.000,B 0.000,C 90.000,E1 261.951} C_DIS
LIN {X 0.084,Y -637.780,Z 332.247,A 0.000,B 0.000,C 90.000,E1 260.443} C_DIS
LIN {X 0.197,Y -640.133,Z 332.234,A 0.000,B 0.000,C 90.000,E1 258.173} C_DIS
LIN {X 0.328,Y -642.385,Z 332.225,A 0.000,B 0.000,C 90.000,E1 256.408} C_DIS
LIN {X -0.286,Y -643.645,Z 332.219,A 0.000,B 0.000,C 90.000,E1 255.463} C_DIS
LIN {X -0.118,Y -644.366,Z 332.215,A 0.000,B 0.000,C 90.000,E1 254.700} C_DIS
LIN {X -0.070,Y -645.326,Z 332.208,A 0.000,B 0.000,C 90.000,E1 253.449} C_DIS
LIN {X 0.182,Y -645.944,Z 332.201,A 0.000,B 0.000,C 90.000,E1 252.181} C_DIS
LIN {X 0.083,Y -646.135,Z 332.198,A 0.000,B 0.000,C 90.000,E1 251.692} C_DIS
LIN {X -0.161,Y -646.023,Z 332.194,A 0.000,B 0.000,C 90.000,E1 250.967} C_DIS
LIN {X 0.356,Y -645.831,Z 332.191,A 0.000,B 0.000,C 90.000,E1 250.423} C_DIS
LIN {X 0.263,Y -645.459,Z 332.189,A 0.000,B 0.000,C 90.000,E1 249.934} C_DIS
LIN {X 0.006,Y -644.640,Z 332.185,A 0.000,B 0.000,C 90.000,E1 249.209} C_DIS
LIN {X -0.096,Y -643.940,Z 332.182,A 0.000,B 0.000,C 90.000,E1 248.720} C_DIS
LIN {X -0.140,Y -642.676,Z 332.178,A 0.000,B 0.000,C 90.000,E1 247.975} C_DIS
LIN {X -0.131,Y -640.614,Z 332.172,A 0.000,B 0.000,C 90.000,E1 246.975} C_DIS
LIN {X -0.146,Y -638.121,Z 332.167,A 0.000,B 0.000,C 90.000,E1 245.973} C_DIS
LIN {X -0.196,Y -635.424,Z 332.161,A 0.000,B 0.000,C 90.000,E1 244.973} C_DIS
LIN {X -0.014,Y -632.275,Z 332.155,A 0.000,B 0.000,C 90.000,E1 243.948} C_DIS
LIN {X 0.127,Y -628.872,Z 332.150,A 0.000,B 0.000,C 90.000,E1 242.922} C_DIS
LIN {X 0.232,Y -624.516,Z 332.143,A 0.000,B 0.000,C 90.000,E1 241.641} C_DIS
LIN {X 0.006,Y -619.285,Z 332.134,A 0.000,B 0.000,C 90.000,E1 240.127} C_DIS
LIN {X -0.008,Y -614.007,Z 332.126,A 0.000,B 0.000,C 90.000,E1 238.584} C_DIS
LIN {X -0.076,Y -609.615,Z 332.118,A 0.000,B 0.000,C 90.000,E1 237.296} C_DIS
LIN {X -0.221,Y -605.094,Z 332.111,A 0.000,B 0.000,C 90.000,E1 236.008} C_DIS
LIN {X 0.029,Y -598.641,Z 332.101,A 0.000,B 0.000,C 90.000,E1 234.149} C_DIS
LIN {X -0.343,Y -594.971,Z 332.095,A 0.000,B 0.000,C 90.000,E1 233.130} C_DIS
LIN {X 0.080,Y -591.079,Z 332.089,A 0.000,B 0.000,C 90.000,E1 232.029} C_DIS
LIN {X 0.012,Y -585.393,Z 332.080,A 0.000,B 0.000,C 90.000,E1 230.436} C_DIS
LIN {X 0.017,Y -580.783,Z 332.073,A 0.000,B 0.000,C 90.000,E1 229.094} C_DIS
LIN {X -0.250,Y -574.504,Z 332.062,A 0.000,B 0.000,C 90.000,E1 227.229} C_DIS
LIN {X -0.180,Y -570.893,Z 332.056,A 0.000,B 0.000,C 90.000,E1 226.134} C_DIS
LIN {X 0.106,Y -564.595,Z 332.046,A 0.000,B 0.000,C 90.000,E1 224.190} C_DIS
LIN {X -0.083,Y -557.440,Z 332.033,A 0.000,B 0.000,C 90.000,E1 222.000} C_DIS
LIN {X -0.069,Y -550.333,Z 332.021,A 0.000,B 0.000,C 90.000,E1 219.769} C_DIS
LIN {X 0.144,Y -546.896,Z 332.015,A 0.000,B 0.000,C 90.000,E1 218.624} C_DIS
LIN {X 0.011,Y -540.079,Z 332.002,A 0.000,B 0.000,C 90.000,E1 216.377} C_DIS
LIN {X -0.208,Y -535.286,Z 331.993,A 0.000,B 0.000,C 90.000,E1 214.692} C_DIS
LIN {X -0.110,Y -529.882,Z 331.982,A 0.000,B 0.000,C 90.000,E1 212.673} C_DIS
LIN {X 0.131,Y -524.325,Z 331.969,A 0.000,B 0.000,C 90.000,E1 210.335} C_DIS
LIN {X 0.219,Y -520.955,Z 331.961,A 0.000,B 0.000,C 90.000,E1 208.871} C_DIS
LIN {X -0.222,Y -516.274,Z 331.949,A 0.000,B 0.000,C 90.000,E1 206.873} C_DIS
LIN {X -0.084,Y -513.040,Z 331.941,A 0.000,B 0.000,C 90.000,E1 205.387} C_DIS
LIN {X 0.020,Y -509.798,Z 331.933,A 0.000,B 0.000,C 90.000,E1 203.898} C_DIS
LIN {X -0.023,Y -507.157,Z 331.926,A 0.000,B 0.000,C 90.000,E1 202.717} C_DIS
LIN {X 0.155,Y -502.471,Z 331.915,A 0.000,B 0.000,C 90.000,E1 200.610} C_DIS
LIN {X -0.182,Y -499.802,Z 331.908,A 0.000,B 0.000,C 90.000,E1 199.450} C_DIS
LIN {X -0.086,Y -495.250,Z 331.896,A 0.000,B 0.000,C 90.000,E1 197.330} C_DIS
LIN {X 0.070,Y -491.004,Z 331.884,A 0.000,B 0.000,C 90.000,E1 195.190} C_DIS
LIN {X -0.003,Y -487.008,Z 331.873,A 0.000,B 0.000,C 90.000,E1 193.063} C_DIS
LIN {X -0.035,Y -484.236,Z 331.864,A 0.000,B 0.000,C 90.000,E1 191.535} C_DIS
LIN {X -0.219,Y -481.544,Z 331.856,A 0.000,B 0.000,C 90.000,E1 190.018} C_DIS
LIN {X -0.208,Y -478.388,Z 331.845,A 0.000,B 0.000,C 90.000,E1 188.163} C_DIS
LIN {X -0.029,Y -474.985,Z 331.833,A 0.000,B 0.000,C 90.000,E1 185.967} C_DIS
LIN {X -0.012,Y -471.105,Z 331.818,A 0.000,B 0.000,C 90.000,E1 183.154} C_DIS
LIN {X 0.092,Y -466.367,Z 331.793,A 0.000,B 0.000,C 90.000,E1 178.740} C_DIS
LIN {X 0.049,Y -463.914,Z 331.772,A 0.000,B 0.000,C 90.000,E1 174.951} C_DIS
LIN {X 0.048,Y -463.127,Z 331.754,A 0.000,B 0.000,C 90.000,E1 171.781} C_DIS
LIN {X 0.195,Y -463.110,Z 331.744,A 0.000,B 0.000,C 90.000,E1 169.859} C_DIS
LIN {X 0.045,Y -464.091,Z 331.721,A 0.000,B 0.000,C 90.000,E1 165.755} C_DIS
LIN {X -0.116,Y -465.279,Z 331.709,A 0.000,B 0.000,C 90.000,E1 163.559} C_DIS
LIN {X -0.022,Y -468.770,Z 331.686,A 0.000,B 0.000,C 90.000,E1 159.444} C_DIS
LIN {X -0.028,Y -472.700,Z 331.668,A 0.000,B 0.000,C 90.000,E1 156.305} C_DIS
LIN {X -0.126,Y -476.709,Z 331.655,A 0.000,B 0.000,C 90.000,E1 153.819} C_DIS
LIN {X 0.107,Y -482.204,Z 331.639,A 0.000,B 0.000,C 90.000,E1 151.001} C_DIS
LIN {X -0.085,Y -487.086,Z 331.627,A 0.000,B 0.000,C 90.000,E1 148.869} C_DIS
LIN {X 0.115,Y -492.607,Z 331.615,A 0.000,B 0.000,C 90.000,E1 146.707} C_DIS
LIN {X -0.085,Y -498.439,Z 331.603,A 0.000,B 0.000,C 90.000,E1 144.609} C_DIS
LIN {X 0.276,Y -503.527,Z 331.593,A 0.000,B 0.000,C 90.000,E1 142.763} C_DIS
LIN {X -0.163,Y -506.811,Z 331.587,A 0.000,B 0.000,C 90.000,E1 141.618} C_DIS
LIN {X -0.148,Y -509.024,Z 331.582,A 0.000,B 0.000,C 90.000,E1 140.723} C_DIS
LIN {X -0.198,Y -511.878,Z 331.575,A 0.000,B 0.000,C 90.000,E1 139.542} C_DIS
LIN {X 0.039,Y -514.947,Z 331.567,A 0.000,B 0.000,C 90.000,E1 138.038} C_DIS
LIN {X 0.104,Y -516.459,Z 331.562,A 0.000,B 0.000,C 90.000,E1 137.148} C_DIS
LIN {X -0.081,Y -517.279,Z 331.559,A 0.000,B 0.000,C 90.000,E1 136.581} C_DIS
LIN {X 0.032,Y -518.141,Z 331.554,A 0.000,B 0.000,C 90.000,E1 135.688} C_DIS
LIN {X 0.055,Y -518.829,Z 331.547,A 0.000,B 0.000,C 90.000,E1 134.514} C_DIS
LIN {X 0.173,Y -519.057,Z 331.543,A 0.000,B 0.000,C 90.000,E1 133.623} C_DIS
LIN {X 0.004,Y -519.058,Z 331.539,A 0.000,B 0.000,C 90.000,E1 133.056} C_DIS
LIN {X 0.148,Y -518.760,Z 331.534,A 0.000,B 0.000,C 90.000,E1 132.162} C_DIS
LIN {X -0.090,Y -518.133,Z 331.529,A 0.000,B 0.000,C 90.000,E1 131.310} C_DIS
LIN {X 0.323,Y -516.847,Z 331.523,A 0.000,B 0.000,C 90.000,E1 130.092} C_DIS
LIN {X -0.274,Y -515.723,Z 331.518,A 0.000,B 0.000,C 90.000,E1 129.277} C_DIS
LIN {X -0.063,Y -513.325,Z 331.508,A 0.000,B 0.000,C 90.000,E1 127.488} C_DIS
LIN {X 0.036,Y -511.627,Z 331.502,A 0.000,B 0.000,C 90.000,E1 126.297} C_DIS
LIN {X 0.028,Y -509.312,Z 331.493,A 0.000,B 0.000,C 90.000,E1 124.818} C_DIS
LIN {X 0.070,Y -507.151,Z 331.487,A 0.000,B 0.000,C 90.000,E1 123.627} C_DIS
LIN {X 0.111,Y -504.337,Z 331.479,A 0.000,B 0.000,C 90.000,E1 122.133} C_DIS
LIN {X 0.002,Y -499.996,Z 331.467,A 0.000,B 0.000,C 90.000,E1 120.050} C_DIS
LIN {X -0.161,Y -496.733,Z 331.459,A 0.000,B 0.000,C 90.000,E1 118.565} C_DIS
LIN {X -0.075,Y -492.104,Z 331.447,A 0.000,B 0.000,C 90.000,E1 116.437} C_DIS
LIN {X 0.089,Y -488.077,Z 331.437,A 0.000,B 0.000,C 90.000,E1 114.591} C_DIS
LIN {X -0.061,Y -484.558,Z 331.428,A 0.000,B 0.000,C 90.000,E1 113.078} C_DIS
LIN {X -0.023,Y -480.278,Z 331.418,A 0.000,B 0.000,C 90.000,E1 111.227} C_DIS
LIN {X -0.055,Y -477.140,Z 331.411,A 0.000,B 0.000,C 90.000,E1 109.993} C_DIS
LIN {X 0.175,Y -474.790,Z 331.406,A 0.000,B 0.000,C 90.000,E1 109.033} C_DIS
LIN {X -0.065,Y -472.342,Z 331.401,A 0.000,B 0.000,C 90.000,E1 108.127} C_DIS
LIN {X 0.066,Y -468.941,Z 331.394,A 0.000,B 0.000,C 90.000,E1 106.858} C_DIS
LIN {X 0.071,Y -465.736,Z 331.387,A 0.000,B 0.000,C 90.000,E1 105.717} C_DIS
LIN {X 0.031,Y -465.744,Z 331.387,A 0.000,B 0.000,C 90.000,E1 105.717} C_DIS
LIN {X 0.182,Y -467.585,Z 331.383,A 0.000,B 0.000,C 90.000,E1 104.954} C_DIS
LIN {X -0.085,Y -468.587,Z 331.380,A 0.000,B 0.000,C 90.000,E1 104.356} C_DIS
LIN {X 0.142,Y -475.814,Z 331.357,A 0.000,B 0.000,C 90.000,E1 100.254} C_DIS
LIN {X -0.021,Y -476.311,Z 331.355,A 0.000,B 0.000,C 90.000,E1 99.962} C_DIS
LIN {X -0.073,Y -481.799,Z 331.331,A 0.000,B 0.000,C 90.000,E1 95.625} C_DIS
LIN {X -0.226,Y -482.173,Z 331.330,A 0.000,B 0.000,C 90.000,E1 95.334} C_DIS
LIN {X 0.188,Y -485.314,Z 331.306,A 0.000,B 0.000,C 90.000,E1 90.974} C_DIS
LIN {X 0.012,Y -485.536,Z 331.304,A 0.000,B 0.000,C 90.000,E1 90.688} C_DIS
LIN {X 0.220,Y -486.322,Z 331.282,A 0.000,B 0.000,C 90.000,E1 86.674} C_DIS
LIN {X -0.131,Y -486.301,Z 331.278,A 0.000,B 0.000,C 90.000,E1 86.102} C_DIS
LIN {X 0.074,Y -484.695,Z 331.254,A 0.000,B 0.000,C 90.000,E1 81.781} C_DIS
LIN {X -0.058,Y -484.592,Z 331.253,A 0.000,B 0.000,C 90.000,E1 81.489} C_DIS
LIN {X -0.177,Y -480.528,Z 331.227,A 0.000,B 0.000,C 90.000,E1 76.881} C_DIS
LIN {X -0.093,Y -477.364,Z 331.216,A 0.000,B 0.000,C 90.000,E1 74.810} C_DIS
LIN {X -0.134,Y -477.376,Z 331.216,A 0.000,B 0.000,C 90.000,E1 74.810} C_DIS
LIN {X -0.254,Y -479.889,Z 331.212,A 0.000,B 0.000,C 90.000,E1 74.102} C_DIS
LIN {X 0.005,Y -483.945,Z 331.205,A 0.000,B 0.000,C 90.000,E1 72.834} C_DIS
LIN {X 0.185,Y -487.611,Z 331.198,A 0.000,B 0.000,C 90.000,E1 71.583} C_DIS
LIN {X 0.137,Y -492.001,Z 331.189,A 0.000,B 0.000,C 90.000,E1 70.061} C_DIS
LIN {X 0.170,Y -496.377,Z 331.181,A 0.000,B 0.000,C 90.000,E1 68.539} C_DIS
LIN {X 0.000,Y -500.758,Z 331.173,A 0.000,B 0.000,C 90.000,E1 67.050} C_DIS
LIN {X -0.176,Y -506.745,Z 331.161,A 0.000,B 0.000,C 90.000,E1 64.973} C_DIS
LIN {X 0.048,Y -511.005,Z 331.153,A 0.000,B 0.000,C 90.000,E1 63.461} C_DIS
